# B&R Automation Studio project A2019059_Linka_Power_CP (part 59)

#### Main.st - Cyclic code
```iecst
//******************************************************************************************************
//	Cylic task for recipe management
//
//	Error numbers:
//	50100  Recipe name parameter is empty
//	50101  Recipe name already exists
//	50102  Recipe name was not found
//  50103  One or more recipe names exceeds maximum length
//	50110  Device name parameter is empty
//	50120  Variable name parameter is empty
//  50130  Recipe management is not initialized
//  50200  Maximum number of recipes reached
//  50300  Task name is incorrect
//  50310  Global recipe structure is incorrect
//******************************************************************************************************

//******************************************************************************************************
// Cyclic task
//******************************************************************************************************

PROGRAM _INIT
		// ----------------------------------------------------------------------------------------
	// The following settings can be adjusted
	Recipe_01.PAR.RecipeVariable 	:= 'RecipeData';		// Top variable structure with recipe data
	Recipe_01.PAR.DeviceName 	:= 'HDD_Receptury';		// Device name from the CPU configuration for X20CPU

	// ----------------------------------------------------------------------------------------
	this							:= 'Recipe_01';			// Name of the global variable structure and this task name
	Recipe_01.PAR.RecipeDirectory 	:= 'Receptury';		        	// Directory where the recipes are stored
	IF(REC_RECIPE_TYPE = typeCSV) THEN
		Recipe_01.PAR.MpLink 		:= gRecipeCsv; 		// MpLink from mappRecipe configuration in physical view
	ELSE
		Recipe_01.PAR.MpLink 		:= gRecipeXml; 		// MpLink from mappRecipe configuration in physical view
	END_IF

	// ----------------------------------------------------------------------------------------
	// Dont change anything below this line
	// ----------------------------------------------------------------------------------------

	// ----------------------------------------------------------------------------------------
	// Make sure global variable structure and task name are correct
	taskStatus := ST_ident(ADR(this), taskGroup, ADR(taskID));
	pvStatus := PV_xgetadr(ADR(this), ADR(pvADR), ADR(pvLEN));
	// Connect global and local structure
	IF(pvStatus = 0) THEN
		RECIPE ACCESS pvADR;
		brsmemset(ADR(RECIPE.ERR), 0 , SIZEOF(RECIPE.ERR));
		RECIPE.PAR.Initialized := FALSE;
	END_IF
	RecipeData;

END_PROGRAM

PROGRAM _CYCLIC
	// --------------------------------------------------------------------------------------------------------------------
	// Make sure task name and global structure correct
	IF(pvStatus <> 0) THEN
		RETURN;
	END_IF
	IF(taskStatus <> 0) THEN
		rec_state := CreateError(ADR(RECIPE), ERR_REC_TASK_NAME, "Meno tasku nieje spravne", rec_state);
		RETURN;
	END_IF

	// --------------------------------------------------------------------------------------------------------------------
	// Make sure we dont exceed maximum number of web clients
	IF(RECIPE.PAR.VisuSlotID > REC_MAX_CLIENTS_ID) THEN
		rec_state := CreateError(ADR(RECIPE), ERR_REC_TOO_MANY_CLIENTS, "More than 3 clients try to connect to recipe managment", rec_state);
		RETURN;
	END_IF

	// --------------------------------------------------------------------------------------------------------------------
	// Cyclic function calls
	MpRecipeCsv_0();
	MpRecipeXml_0();

	//**************************************************************************************************
	// Recipe managment state machine
	//**************************************************************************************************
	CASE rec_state OF
		//**********************************************************************************************
		// Wait for command
		//**********************************************************************************************
		REC_WAIT:
			// --------------------------------------------------------------------------------------------------------------------
			// Track filter change and data refresh
			IF ((brwcscmp(ADR(RecipeFilterOld[VisuSlotID]), ADR(RECIPE.VIS[VisuSlotID].RecipeFilter)) <> 0) OR (RecipeNumOld[VisuSlotID] <> RECIPE.DAT.RecipeNum)) THEN
				brsmemset(ADR(RECIPE.VIS[VisuSlotID].RecipeNames), 0, SIZEOF(RECIPE.VIS[VisuSlotID].RecipeNames));
				idy := 0;
				IF(RECIPE.DAT.RecipeNum > 0) THEN
					FOR idx:=0 TO RECIPE.DAT.RecipeNum - 1 DO
						// --------------------------------------------------------------------------------
						// Verify that file name contains filter
						IF (brwcslen(ADR(RECIPE.VIS[VisuSlotID].RecipeFilter)) = 0 OR IsInstrW(ADR(RECIPE.DAT.RecipeNames[idx]), ADR(RECIPE.VIS[VisuSlotID].RecipeFilter))) THEN
							WString2DataProvider(ADR(RECIPE.DAT.RecipeNames[idx]), ADR(tmpWStr1));
							RECIPE.VIS[VisuSlotID].RecipeNames[idy] := tmpWStr1;
							idy := idy + 1;
						END_IF
					END_FOR;
					brwcscpy(ADR(RecipeFilterOld[VisuSlotID]), ADR(RECIPE.VIS[VisuSlotID].RecipeFilter));
				END_IF
				RecipeNumOld[VisuSlotID] := RECIPE.DAT.RecipeNum;
				RECIPE.VIS[VisuSlotID].RecipeNum := idy;
			END_IF
			// Cylce through the client web seesions
			VisuSlotID := VisuSlotID + 1;
			IF(VisuSlotID > REC_MAX_CLIENTS_ID) THEN
				VisuSlotID := 0;
			END_IF

			// --------------------------------------------------------------------------------------------------------------------
			// Disable buttons in visualization when number of recipes is 0
			IF(RECIPE.DAT.RecipeNum = 0) THEN
				RECIPE.PAR.VisuEnableCommand := FALSE;
			ELSE
				RECIPE.PAR.VisuEnableCommand := TRUE;
			END_IF

			// ----------------------------------------------------------------------------------------
			// Reset error reset
			MpRecipeCsv_0.ErrorReset := FALSE;
			MpRecipeXml_0.ErrorReset := FALSE;
			MpRecipeRegPar_0.ErrorReset := FALSE;

			// ----------------------------------------------------------------------------------------
			// Command refresh
			IF (RECIPE.CMD.Init = TRUE) THEN
				// Reset data structure and trigger name refresh for vis
				brsmemset(ADR(RECIPE.DAT), 0, SIZEOF(RECIPE.DAT));
				brsmemset(ADR(RecipeIDs), 0, SIZEOF(RecipeIDs));
				brsmemset(ADR(RecipeNumOld), 16#FF, SIZEOF(RecipeNumOld));
				// Skip variable binding if already initialized
				IF(MpRecipeRegPar_1.PVName <> 0) THEN
					rec_state := REC_READ_DIR;
				ELSE
					// Register recipe name varibale first if unicode is used
					IF(REC_USE_UNICODE) THEN
						rec_state := REC_REG_NAME;
					ELSE
						rec_state := REC_REG_VAR;
					END_IF
				END_IF
				MpRecipeRegPar_1.Enable := FALSE;
				// ----------------------------------------------------------------------------------------
				// Command new recipe
			ELSIF (RECIPE.CMD.New = TRUE AND RECIPE.PAR.RecipeName <> "") THEN
				// Show current state
				animation := WorkingStatus(ADR(RECIPE), ADR("Vytvaram recepturu..."), animation);
				// Verify that we still have space in list
				IF (RECIPE.DAT.RecipeNum > REC_MAX_NUM) THEN
					rec_state := CreateError(ADR(RECIPE), ERR_REC_MAX_NUM, "Maximalny pocet receptur dosiahnuty", rec_state);
					RETURN;
				END_IF
				// Make sure recipe does not already exist
				IF(FindRecName(ADR(RECIPE), RECIPE.PAR.RecipeName) <> REC_DOES_NOT_EXIST) THEN
					tmpWStr1 := "Nazov raceptury ";
					brwcscat(ADR(tmpWStr1), ADR(RECIPE.PAR.RecipeName));
					brwcscat(ADR(tmpWStr1), ADR(" uz existuje"));
					rec_state := CreateError(ADR(RECIPE), ERR_REC_NAME_EXISTS, tmpWStr1, rec_state);
					RETURN;
				END_IF
				// Turn on variable saving, reset selected recipe, copy recipe name to local variable
				MpRecipeRegPar_1.Enable := TRUE;;
				RECIPE.VIS[RECIPE.PAR.VisuSlotID].RecipeSelect := "";
				rec_state := REC_GEN_FILE_NAME;
				// ----------------------------------------------------------------------------------------
				// Command load recipe
			ELSIF (RECIPE.CMD.Load = TRUE AND RECIPE.PAR.RecipeName <> "") THEN
				// Show current state
				animation := WorkingStatus(ADR(RECIPE), ADR("Nahravam recepturu..."), animation);
				// Turn on variable saving, copy recipe name to local variable
				MpRecipeRegPar_1.Enable := TRUE;;
				rec_state := REC_GEN_FILE_NAME;
				// ----------------------------------------------------------------------------------------
				// Command load recipe
			ELSIF (RECIPE.CMD.Save = TRUE AND (RECIPE.PAR.RecipeName <> "" OR RECIPE.PAR.RecipeNameNew <> "")) THEN
				// Show current state
				animation := WorkingStatus(ADR(RECIPE), ADR("Ukladam recepturu..."), animation);
				IF(RECIPE.PAR.RecipeName = "") THEN
					RECIPE.PAR.RecipeName := RECIPE.PAR.RecipeNameNew;
				END_IF
				// Turn on variable saving, copy recipe name to local variable
				MpRecipeRegPar_1.Enable := TRUE;;
				rec_state := REC_GEN_FILE_NAME;
				// ----------------------------------------------------------------------------------------
				// Command delete recipe
			ELSIF (RECIPE.CMD.Delete = TRUE AND RECIPE.PAR.RecipeName <> "") THEN
				// Show current state, copy recipe name to local variable
				animation := WorkingStatus(ADR(RECIPE), ADR("Mazem recepturu..."), animation);
				rec_state := REC_GEN_FILE_NAME;
				// ----------------------------------------------------------------------------------------
				// Rename recipe
			ELSIF (RECIPE.CMD.Rename = TRUE AND RECIPE.PAR.RecipeName <> "" AND RECIPE.PAR.RecipeNameNew <> "") THEN
				// Show current state
				animation := WorkingStatus(ADR(RECIPE), ADR("Premenovavam recepturu..."), animation);
				// Make sure new recipe name does not already exist
				IF(FindRecName(ADR(RECIPE), RECIPE.PAR.RecipeNameNew) <> REC_DOES_NOT_EXIST) THEN
					tmpWStr1 := "Nove meno receptury ";
					brwcscat(ADR(tmpWStr1), ADR(RECIPE.PAR.RecipeNameNew));
					brwcscat(ADR(tmpWStr1), ADR(" uz existuje"));
					rec_state := CreateError(ADR(RECIPE), ERR_REC_NAME_EXISTS, tmpWStr1, rec_state);
					RETURN;
				END_IF
				// Turn on variable saving, reset selected recipe, copy recipe name to local variable
				MpRecipeRegPar_1.Enable := TRUE;
				brsmemset(ADR(RecipeNumOld), 16#FF, SIZEOF(RecipeNumOld));
				RECIPE.VIS[RECIPE.PAR.VisuSlotID].RecipeSelect := "";
				RecipeNameNew := RECIPE.PAR.RecipeNameNew;
				rec_state := REC_GEN_FILE_NAME;
			END_IF
			RecipeName := RECIPE.PAR.RecipeName;

			// ----------------------------------------------------------------------------------------
			// Check parameters
			IF (RECIPE.CMD.Init OR RECIPE.CMD.New OR RECIPE.CMD.Load OR RECIPE.CMD.Save OR RECIPE.CMD.Rename OR RECIPE.CMD.Delete) THEN
				// Make sure recipe mangament was intialized
				IF (NOT RECIPE.CMD.Init AND NOT RECIPE.PAR.Initialized) THEN
					rec_state := CreateError(ADR(RECIPE), ERR_REC_NOT_INITIALIZED, "Receptury nie su zinicializovane", rec_state);
				END_IF
				// Make sure recipe name is valid
				IF((RECIPE.CMD.New OR RECIPE.CMD.Load OR RECIPE.CMD.Save OR RECIPE.CMD.Rename OR RECIPE.CMD.Delete) AND RecipeName = "") THEN
					rec_state := CreateError(ADR(RECIPE), ERR_REC_NAME_EMPTY, "Meno receptury je prazdne", rec_state);
				END_IF
				// Make sure new recipe name is valid
				IF((RECIPE.CMD.Rename) AND RecipeNameNew = "") THEN
					rec_state := CreateError(ADR(RECIPE), ERR_REC_NAME_EMPTY, "Nova receptura je prazdna", rec_state);
				END_IF
				// Make sure device name is valid
				IF(RECIPE.PAR.DeviceName = '') THEN
					rec_state := CreateError(ADR(RECIPE), ERR_REC_DEV_NAME_EMPTY, "Meno zariadenia je prazdne", rec_state);
				END_IF
				// Make sure variable name is valid
				IF(RECIPE.PAR.RecipeVariable = '') THEN
					rec_state := CreateError(ADR(RECIPE), ERR_REC_VAR_NAME_EMPTY, "Meno premennej je prazdne", rec_state);
				END_IF

				RECIPE.PAR.VisuEnableCommand := FALSE;
			END_IF
			//**********************************************************************************************
			// Register recipe name
			//**********************************************************************************************
		REC_REG_NAME:
			// Generate string for local recipe name
			tmpStr1 := this;
			brsstrcat(ADR(tmpStr1), ADR(':RecipeName'));

			MpRecipeRegPar_0.Enable := TRUE;
			MpRecipeRegPar_0.MpLink := ADR(RECIPE.PAR.MpLink);
			MpRecipeRegPar_0.PVName := ADR(tmpStr1);

			// ----------------------------------------------------------------------------------------
			// OK
			IF (NOT MpRecipeRegPar_0.Active AND NOT MpRecipeRegPar_0.Error) THEN
				rec_state := REC_REG_VAR;
				// Error
			ELSIF (MpRecipeRegPar_0.Error) THEN
				rec_state := CreateError(ADR(RECIPE), MpRecipeRegPar_0.StatusID, "Error trying to register recipe name", rec_state);
			END_IF
			//**********************************************************************************************
			// Register variable structure
			//**********************************************************************************************
		REC_REG_VAR:
			MpRecipeRegPar_1.MpLink := ADR(RECIPE.PAR.MpLink);
			MpRecipeRegPar_1.PVName := ADR(RECIPE.PAR.RecipeVariable);

			// ----------------------------------------------------------------------------------------
			// OK
			IF (NOT MpRecipeRegPar_1.Active AND NOT MpRecipeRegPar_1.Error) THEN
				rec_state := REC_CREATE_DIR;
				// Error
			ELSIF (MpRecipeRegPar_1.Error) THEN
				tmpWStr1 := "Error trying to register variable name ";
				brwcsconv(ADR(tmpWStr2), ADR(RECIPE.PAR.RecipeVariable), brwU8toUC);
				brwcscat(ADR(tmpWStr1), ADR(tmpWStr2));
				rec_state := CreateError(ADR(RECIPE), MpRecipeRegPar_1.StatusID, tmpWStr1, rec_state);
			END_IF
			//**********************************************************************************************
			// Create recipe directory
			//**********************************************************************************************
		REC_CREATE_DIR:
			DCreate.enable 	:= 1;
			DCreate.pDevice	:= ADR(RECIPE.PAR.DeviceName);
			DCreate.pName := ADR(RECIPE.PAR.RecipeDirectory);
			DCreate();

			// ----------------------------------------------------------------------------------------
			// OK
			IF (DCreate.status = OK OR DCreate.status = fiERR_DIR_ALREADY_EXIST) THEN
				// Reset command and return to wait state
				rec_state := REC_READ_DIR;
				// Error
			ELSIF (DCreate.status <> ERR_FUB_BUSY) THEN
				rec_state := CreateError(ADR(RECIPE), DCreate.status, "Porucha vytvorenia adresara", rec_state);
			END_IF
			//**********************************************************************************************
			// Read directory information
			//**********************************************************************************************
		REC_READ_DIR:
			// Show current state
			animation := WorkingStatus(ADR(RECIPE), ADR("Nacitavam recepturu..."), animation);
			// ----------------------------------------------------------------------------------------
			// Clear all entrys
			brsmemset(ADR(RECIPE.DAT), 0, SIZEOF(RECIPE.DAT));
			RECIPE.DAT.RecipeNum := 0;
			// ----------------------------------------------------------------------------------------
			// Set values and get device dir
			DInfo.enable 	:= 1;
			DInfo.pDevice	:= ADR(RECIPE.PAR.DeviceName);
			DInfo();

			// ----------------------------------------------------------------------------------------
			// OK
			IF (DInfo.status = OK) THEN
				rec_state := REC_READ_DIR_1;
			ELSIF (DInfo.status = fiERR_DEVICE_MANAGER) THEN
				tmpWStr1 := "Suborovy system ";
				brwcsconv(ADR(tmpWStr2), ADR(RECIPE.PAR.DeviceName), brwU8toUC);
				brwcscat(ADR(tmpWStr1), ADR(tmpWStr2));
				brwcscat(ADR(tmpWStr1), ADR(" je nedostupny"));
				rec_state := CreateError(ADR(RECIPE), DInfo.status, tmpWStr1, rec_state);
			ELSIF (DInfo.status = fiERR_DIR_NOT_EXIST) THEN
				tmpWStr1 := "Subor ";
				brwcsconv(ADR(tmpWStr2), ADR(RECIPE.PAR.RecipeDirectory), brwU8toUC);
				brwcscat(ADR(tmpWStr1), ADR(tmpWStr2));
				brwcscat(ADR(tmpWStr1), ADR(" je nedostupny"));
				rec_state := CreateError(ADR(RECIPE), DInfo.status, tmpWStr1, rec_state);
				// Error
			ELSIF (DInfo.status <> ERR_FUB_BUSY) THEN
				rec_state := CreateError(ADR(RECIPE), DInfo.status, "Error dir info", rec_state);
			END_IF
			//**********************************************************************************************
			// Open directory
			//**********************************************************************************************
		REC_READ_DIR_1:
			DOpen.enable 	:= 1;
			DOpen.pDevice	:= ADR(RECIPE.PAR.DeviceName);
			DOpen.pName 	:= ADR(RECIPE.PAR.RecipeDirectory);
			DOpen();

			// ----------------------------------------------------------------------------------------
			// OK
			IF (DOpen.status = OK) THEN
				rec_state := REC_READ_DIR_2;
			ELSIF (DInfo.status = fiERR_DIR_NOT_EXIST) THEN
				tmpWStr1 := "Adresar ";
				brwcsconv(ADR(tmpWStr2), ADR(RECIPE.PAR.RecipeDirectory), brwU8toUC);
				brwcscat(ADR(tmpWStr1), ADR(tmpWStr2));
				brwcscat(ADR(tmpWStr1), ADR(" je nedostupny"));
				rec_state := CreateError(ADR(RECIPE), DInfo.status, tmpWStr1, rec_state);
				// Error
			ELSIF (DOpen.status <> ERR_FUB_BUSY) THEN
				rec_state := CreateError(ADR(RECIPE), DOpen.status, "Porucha otvorenie adresara", rec_state);
			END_IF;
			//**********************************************************************************************
			// Read file directory information
			//**********************************************************************************************
		REC_READ_DIR_2:
			DRead.enable 	:= 1;
			DRead.ident		:= DOpen.ident;
			DRead.pData 	:= ADR(lDirReadData);
			DRead.data_len 	:= SIZEOF(lDirReadData);
			DRead();

			// ----------------------------------------------------------------------------------------
			// OK
			IF (DRead.status = OK AND lDirReadData.Mode = fiFILE) THEN
				animation := WorkingStatus(ADR(RECIPE), ADR("Inicializacia receptur..."), animation);
				// Make sure file name does not exceed maximum string size
				IF (brsstrlen(ADR(lDirReadData.Filename)) < REC_NAME_LENGTH) THEN
					// Copy dir info to string
					brsmemset(ADR(RECIPE.PAR.RecipeID), 0, SIZEOF(RECIPE.PAR.RecipeID));
					brsstrcpy(ADR(RECIPE.PAR.RecipeID), ADR(lDirReadData.Filename));
					// Make sure file extension is CSV or XML
					IF(brsstrlen(ADR(RECIPE.PAR.RecipeID)) > 4 AND ((REC_RECIPE_TYPE = typeCSV AND brsmemcmp(ADR(RECIPE.PAR.RecipeID) + (brsstrlen(ADR(RECIPE.PAR.RecipeID)) - 4), ADR('.csv'), 4) = 0) OR (REC_RECIPE_TYPE = typeXML AND brsmemcmp(ADR(RECIPE.PAR.RecipeID) + (brsstrlen(ADR(RECIPE.PAR.RecipeID)) - 4), ADR('.xml'), 4) = 0))) THEN
						brsmemset(ADR(RECIPE.PAR.RecipeID) + (brsstrlen(ADR(RECIPE.PAR.RecipeID)) - 4), 0, 4);
						// ------------------------------------------------------------------------------------
						// Verify that we still have space in list
						IF (RECIPE.DAT.RecipeNum <= REC_MAX_NUM) THEN
							// --------------------------------------------------------------------
							// Read recipe name from recipe data in next step when using unicode
							IF(REC_USE_UNICODE) THEN
								RecipeIDs[brsatoi(ADR(RECIPE.PAR.RecipeID))] := TRUE;
								rec_state := REC_GEN_FILE_NAME;
								// Generate recipe name from file name
							ELSE
								brwcsconv(ADR(RecipeName), ADR(RECIPE.PAR.RecipeID), brwU8toUC);
								// Generate ASCII data, insert recipe into list
								InsertRecName(ADR(RECIPE), RecipeName, RECIPE.PAR.RecipeID);
							END_IF
							// Error
						ELSE
							rec_state := CreateError(ADR(RECIPE), ERR_REC_MAX_NUM, "Maximalny pocet receptur dosiahnuty", rec_state);
						END_IF
					END_IF
				ELSE
					has_oversized_items := TRUE;
				END_IF
				// Last entry reached
			ELSIF (DRead.status = fiERR_NO_MORE_ENTRIES) THEN
				rec_state := REC_READ_DIR_3;
				// Error
			ELSIF (DRead.status <> ERR_FUB_BUSY AND DRead.status <> OK) THEN
				rec_state := CreateError(ADR(RECIPE), DRead.status, "Porucha citania zoznamu receptur", rec_state);
			END_IF
			//**********************************************************************************************
			// Close directory information
			//**********************************************************************************************
		REC_READ_DIR_3:
			DClose.enable 	:= 1;
			DClose.ident	:= DOpen.ident;
			DClose();

			// ----------------------------------------------------------------------------------------
			// OK
			IF (DClose.status = OK) THEN
				// Reset command and return to wait state
				RECIPE.DAT.Status := "Inicializacia receptur ukoncena";
				RECIPE.CMD.Init	:= 0;
				RECIPE.PAR.RecipeID := '';
				RECIPE.PAR.Initialized := TRUE;
				DClose.ident	:= 0;
				IF(has_oversized_items) THEN
					rec_state := CreateError(ADR(RECIPE), ERR_REC_NAME_LENGTH, "Meno receptury presiahlo maximalny pocet znakov", rec_state);
				ELSE
					rec_state := REC_WAIT;
				END_IF
				// Error
			ELSIF (DClose.status <> ERR_FUB_BUSY) THEN
				rec_state := CreateError(ADR(RECIPE), DClose.status, "Porucha zatvorenia adresara", rec_state);
			END_IF
			//**********************************************************************************************
			// Generate recipe name	full path and file name
			//**********************************************************************************************
		REC_GEN_FILE_NAME:
			// Find recipe entry
			RecipeIndex := FindRecName(ADR(RECIPE), RecipeName);

			// Generate file name when using unicode strings
			IF(REC_USE_UNICODE) THEN
				// Ignore during init process
				IF(NOT RECIPE.CMD.Init) THEN
					// Find empty slot for new recipe
					IF(RECIPE.CMD.New) THEN
						RecipeIndex := 0;
						WHILE (RecipeIDs[RecipeIndex] = TRUE AND RecipeIndex <= REC_MAX_NUM) DO
							RecipeIndex := RecipeIndex + 1;
						END_WHILE;
						// Make sure we found empty slot
						IF(RecipeIndex <= REC_MAX_NUM AND RecipeIDs[RecipeIndex] = FALSE) THEN
							brsitoa(RecipeIndex, ADR(RECIPE.PAR.RecipeID));
						ELSE
							rec_state := CreateError(ADR(RECIPE), ERR_REC_MAX_NUM, "Prazdny slot nenajdeny", rec_state);
							RETURN;
						END_IF
						// Find recipe name in list	for all other command
					ELSE
						// Recipe name was found
						IF(RecipeIndex <> REC_DOES_NOT_EXIST) THEN
							RECIPE.PAR.RecipeID := RECIPE.DAT.RecipeIDs[RecipeIndex];
							// Recipe name was lost
						ELSE
							tmpWStr1 := "Meno receptury nebolo najdene ";
							brwcscat(ADR(tmpWStr1), ADR(RecipeName));
							rec_state := CreateError(ADR(RECIPE), ERR_REC_NAME_LOST, tmpWStr1, rec_state);
							RETURN;
						END_IF
					END_IF
				END_IF
				// Use recipe name as file name when using standard strings
			ELSE
				brwcsconv(ADR(RECIPE.PAR.RecipeID), ADR(RecipeName), brwUCtoU8);
			END_IF

			// Generate recipe path and extension
			RecipeFullFileName := RECIPE.PAR.RecipeDirectory;
			brsstrcat(ADR(RecipeFullFileName), ADR('/'));
			brsstrcat(ADR(RecipeFullFileName), ADR(RECIPE.PAR.RecipeID));

			// Add file extension
			IF(REC_RECIPE_TYPE = typeCSV) THEN
				brsstrcat(ADR(RecipeFullFileName), ADR('.csv'));
			ELSE
				brsstrcat(ADR(RecipeFullFileName), ADR('.xml'));
			END_IF

			// Save recipe under new name
			IF(RECIPE.CMD.Rename) THEN
				RecipeName := RecipeNameNew;
			END_IF

			// Proceed with next step
			IF(RECIPE.CMD.Delete) THEN
				rec_state := REC_DELETE;
			ELSIF(RECIPE.CMD.Rename AND NOT REC_USE_UNICODE) THEN
				rec_state := REC_RENAME;
			ELSE
				rec_state := REC_LOAD_SAVE;
			END_IF
			//**********************************************************************************************
			// Load or save recipe data
			//**********************************************************************************************
		REC_LOAD_SAVE:

			IF(REC_RECIPE_TYPE = typeCSV) THEN
				MpRecipeCsv_0.Enable := TRUE;
				MpRecipeCsv_0.MpLink := ADR(RECIPE.PAR.MpLink);
				MpRecipeCsv_0.DeviceName := ADR(RECIPE.PAR.DeviceName);
				MpRecipeCsv_0.FileName := ADR(RecipeFullFileName);
				MpRecipeCsv_0.Save := RECIPE.CMD.Save OR RECIPE.CMD.New OR RECIPE.CMD.Rename;
				MpRecipeCsv_0.Load := RECIPE.CMD.Load OR RECIPE.CMD.Init;

				MpRecipeDone := MpRecipeCsv_0.CommandDone;
				MpRecipeError := MpRecipeCsv_0.Error;
				MpRecipeStatusID := MpRecipeCsv_0.StatusID;
			ELSE
				MpRecipeXml_0.Enable := TRUE;
				MpRecipeXml_0.MpLink := ADR(RECIPE.PAR.MpLink);
				MpRecipeXml_0.DeviceName := ADR(RECIPE.PAR.DeviceName);
				MpRecipeXml_0.FileName := ADR(RecipeFullFileName);
				MpRecipeXml_0.Save := RECIPE.CMD.Save OR RECIPE.CMD.New OR RECIPE.CMD.Rename;
				MpRecipeXml_0.Load := RECIPE.CMD.Load OR RECIPE.CMD.Init;

				MpRecipeDone := MpRecipeXml_0.CommandDone;
				MpRecipeError := MpRecipeXml_0.Error;
				MpRecipeStatusID := MpRecipeXml_0.StatusID;
			END_IF

			// ----------------------------------------------------------------------------------------
			// OK
			IF (MpRecipeDone AND NOT MpRecipeError AND MpRecipeStatusID = 0) THEN
				// Reset command and return to wait state
				MpRecipeCsv_0.Load := FALSE;
				MpRecipeCsv_0.Save := FALSE;
				MpRecipeXml_0.Load := FALSE;
				MpRecipeXml_0.Save := FALSE;

				// Continue renaming recipe
				IF(RECIPE.CMD.Rename) THEN
					IF(REC_USE_UNICODE) THEN
						// Remove name from recipe list	and add it again
						RemoveRecName(ADR(RECIPE), RecipeIndex);
						InsertRecName(ADR(RECIPE), RecipeName, RECIPE.PAR.RecipeID);

						RECIPE.VIS[RECIPE.PAR.VisuSlotID].RecipeSelect := RecipeName;
						tmpWStr1 := "Receptura bola premenovana";
						RECIPE.CMD.Rename := 0;
					ELSE
						rec_state := REC_DELETE;
						RETURN;
					END_IF
				END_IF
				// Continue reading recipe names
				IF(RECIPE.CMD.Init) THEN
					InsertRecName(ADR(RECIPE), RecipeName, RECIPE.PAR.RecipeID);
					rec_state := REC_READ_DIR_2;
					RETURN;
				END_IF
				// Finish new recipe
				IF(RECIPE.CMD.New) THEN
					IF(REC_USE_UNICODE) THEN
						RecipeIDs[brsatoi(ADR(RECIPE.PAR.RecipeID))] := TRUE;
					END_IF
					InsertRecName(ADR(RECIPE), RecipeName, RECIPE.PAR.RecipeID);
					RECIPE.VIS[RECIPE.PAR.VisuSlotID].RecipeSelect := RecipeName;
					tmpWStr1 := "Receptura bola vytvorena";
					RECIPE.CMD.New	:= FALSE;
				END_IF
				// Finish load recipe
				IF(RECIPE.CMD.Load) THEN
					tmpWStr1 := "Receptura bola nacitana";
					RECIPE.CMD.Load	:= FALSE;
				END_IF
				// Finish save recipe
				IF(RECIPE.CMD.Save) THEN
					tmpWStr1 := "Receptura bola ulozena";
					RECIPE.CMD.Save	:= FALSE;
				END_IF
				// Complete status string
				CreateMessage(ADR(RECIPE.DAT.Status), ADR(tmpWStr1), ADR(RecipeName), RECIPE.PAR.VisuSlotID);
				rec_state := REC_WAIT;
				// Error
			ELSIF (MpRecipeStatusID = mpRECIPE_WRN_LOAD_WITH_WARN) THEN
				rec_state := CreateError(ADR(RECIPE), MpRecipeStatusID, "Warning recipe read/write/new, check PLC logbook for details", rec_state);
			ELSIF (MpRecipeError OR MpRecipeStatusID <> 0) THEN
				tmpWStr1 := "Error recipe read/write/new ";
				brwcscat(ADR(tmpWStr1), ADR(RecipeName));
				rec_state := CreateError(ADR(RECIPE), MpRecipeStatusID, tmpWStr1, rec_state);
			END_IF
			//**********************************************************************************************
			// Delete selected recipe
			//**********************************************************************************************
		REC_DELETE:
			// ----------------------------------------------------------------------------------------
			// Initialize file delete structure
			FDelete.enable		:= 1;
			FDelete.pDevice 	:= ADR(RECIPE.PAR.DeviceName);
			FDelete.pName		:= ADR(RecipeFullFileName);
			FDelete();

			// ----------------------------------------------------------------------------------------
			// OK
			IF (FDelete.status = OK) THEN
				// Remove name from recipe list
				RemoveRecName(ADR(RECIPE), RecipeIndex);
				// Mark recipe ID as free
				IF(REC_USE_UNICODE) THEN
					RecipeIDs[brsatoi(ADR(RECIPE.PAR.RecipeID))] := FALSE;
				END_IF

				CreateMessage(ADR(RECIPE.DAT.Status), ADR("Receptura bola vymazana"), ADR(RecipeName), RECIPE.PAR.VisuSlotID);
				RECIPE.CMD.Delete := 0;
				rec_state := REC_WAIT;
				// Error
			ELSIF (FDelete.status <> ERR_FUB_BUSY) THEN
				tmpWStr1 := "Porucha vymazania receptury ";
				brwcscat(ADR(tmpWStr1), ADR(RecipeName));
				rec_state := CreateError(ADR(RECIPE), FDelete.status, tmpWStr1, rec_state);
			END_IF
			//**********************************************************************************************
			// Rename selected recipe
			//**********************************************************************************************
		REC_RENAME:
			// Generate recipe path and extension
			tmpStr1 := RECIPE.PAR.RecipeDirectory;
			brsstrcat(ADR(tmpStr1), ADR('/'));
			brwcsconv(ADR(tmpStr2), ADR(RecipeNameNew), brwUCtoU8);
			brsstrcat(ADR(tmpStr1), ADR(tmpStr2));

			// Add file extension
			IF(REC_RECIPE_TYPE = typeCSV) THEN
				brsstrcat(ADR(tmpStr1), ADR('.csv'));
			ELSE
				brsstrcat(ADR(tmpStr1), ADR('.xml'));
			END_IF

			// ----------------------------------------------------------------------------------------
			// Initialize file delete structure
			FRename.enable		:= 1;
			FRename.pDevice 	:= ADR(RECIPE.PAR.DeviceName);
			FRename.pName		:= ADR(RecipeFullFileName);
			FRename.pNewName	:= ADR(tmpStr1);
			FRename();

			// ----------------------------------------------------------------------------------------
			// OK
			IF (FRename.status = OK) THEN
				// Remove name from recipe list	and add it again
				brsmemmove(ADR(RECIPE.DAT.RecipeNames[RecipeIndex]),ADR(RECIPE.DAT.RecipeNames[RecipeIndex+1]), (RECIPE.DAT.RecipeNum) * SIZEOF(RECIPE.DAT.RecipeNames[0]));
				brsmemmove(ADR(RECIPE.DAT.RecipeIDs[RecipeIndex]),ADR(RECIPE.DAT.RecipeIDs[RecipeIndex+1]), (RECIPE.DAT.RecipeNum) * SIZEOF(RECIPE.DAT.RecipeIDs[0]));
				RECIPE.DAT.RecipeNum := RECIPE.DAT.RecipeNum - 1;
				InsertRecName(ADR(RECIPE), RecipeNameNew, RECIPE.PAR.RecipeID);

				RECIPE.VIS[RECIPE.PAR.VisuSlotID].RecipeSelect := RecipeNameNew;
				CreateMessage(ADR(RECIPE.DAT.Status), ADR("Receptura bola premenovana"), ADR(RecipeName), RECIPE.PAR.VisuSlotID);
				RECIPE.CMD.Rename := 0;
				rec_state := REC_WAIT;
				// Error
			ELSIF (FRename.status <> ERR_FUB_BUSY) THEN
				tmpWStr1 := "Porucha premenovania receptury ";
				brwcscat(ADR(tmpWStr1), ADR(RecipeName));
				rec_state := CreateError(ADR(RECIPE), FRename.status, tmpWStr1, rec_state);
			END_IF
			// --------------------------------------------------------------------------------------------------------------------
			// Error
			// --------------------------------------------------------------------------------------------------------------------
		REC_ERROR:
			RECIPE.DAT.Status := "Error state triggered on web client ID ";
			tmpWStr1 := DINT_TO_WSTRING(RECIPE.PAR.VisuSlotID);
			brwcscat(ADR(RECIPE.DAT.Status), ADR(tmpWStr1));
			// --------------------------------------------------------------------------------------------------------------------
			// Make sure we dont exceed maximum number of web clients
			IF(RECIPE.PAR.VisuSlotID <= REC_MAX_CLIENTS_ID) THEN
				RECIPE.VIS[RECIPE.PAR.VisuSlotID].ShowMessageBoxError := TRUE;
			END_IF
			// --------------------------------------------------------------------------------------------------------------------
			// Return to idle state
			IF RECIPE.CMD.ErrorReset THEN
				// Reset function blocks
				MpRecipeCsv_0.ErrorReset := TRUE;
				MpRecipeCsv_0.Save := FALSE;
				MpRecipeCsv_0.Load := FALSE;

				MpRecipeXml_0.ErrorReset := TRUE;
				MpRecipeXml_0.Save := FALSE;
				MpRecipeXml_0.Load := FALSE;

				MpRecipeRegPar_0.ErrorReset := TRUE;

				// Reset error structure
				brsmemset(ADR(RECIPE.ERR), 0, SIZEOF(RECIPE.ERR));
				RECIPE.DAT.Status := "";
				RECIPE.CMD.ErrorReset := FALSE;
				RECIPE.VIS[RECIPE.PAR.VisuSlotID].ShowMessageBoxError := FALSE;
				rec_state := REC_WAIT;
			END_IF;
			brsmemset(ADR(RECIPE.CMD), 0, SIZEOF(RECIPE.CMD));
			RETURN;
	END_CASE
	// --------------------------------------------------------------------------------------------------------------------
	// Cyclic function calls
	MpRecipeRegPar_0();
	MpRecipeRegPar_1();
	MpRecipeCsv_0();
	MpRecipeXml_0();

END_PROGRAM

PROGRAM _EXIT
	(* Insert code here *)

END_PROGRAM
```

#### RecipeVariables.var - Local variables
```iecst
(*------------------------------------------------------------------------------------------------------------------------------------------------------------------------------------------------------------------------*)
(*Local constants*)
VAR CONSTANT
	OK : USINT := 0; (*Constant for status OK *)
	REC_DOES_NOT_EXIST : UINT := 65535; (*Constant for record does not exist*)
END_VAR
(*------------------------------------------------------------------------------------------------------------------------------------------------------------------------------------------------------------------------*)
(*Local Variables*)
VAR
	RECIPE : REFERENCE TO recMAIN; (*Local recipe structure*)
	RecipeIDs : ARRAY[0..REC_MAX_NUM] OF BOOL; (*Used with unicode option, keeps tracks of the IDs used*)
	RecipeIndex : UINT; (*Current recipe index*)
	RecipeName : WSTRING[REC_NAME_LENGTH]; (*Local recipe name*)
	RecipeNameNew : WSTRING[REC_NAME_LENGTH]; (*Local recipe new name*)
	RecipeFullFileName : STRING[200]; (*Full recipe name*)
	RecipeFilterOld : ARRAY[0..REC_MAX_CLIENTS_ID] OF WSTRING[REC_NAME_LENGTH]; (*Track filter change *)
	RecipeNumOld : ARRAY[0..REC_MAX_CLIENTS_ID] OF UINT;
	rec_state : recSTATE := REC_WAIT; (*Main step index *)
	animation : USINT := 0; (*Animation for working status	*)
	VisuSlotID : USINT; (*Slot of the visualization that is current used*)
	idx : UINT;
	idy : UINT;
	has_oversized_items : BOOL; (*Indicates that at least one recipe name exceeds the maximum length*)
	tmpStr1 : STRING[200]; (*Temporary string variable *)
	tmpStr2 : STRING[200]; (*Temporary string variable *)
	tmpWStr1 : WSTRING[REC_VIS_LENGTH]; (*Temporary unicode string variable *)
	tmpWStr2 : WSTRING[REC_VIS_LENGTH]; (*Temporary unicode string variable *)
	lDirReadData : fiDIR_READ_EX_DATA; (*File information structure*)
	this : STRING[100]; (*Name of the task and global recipe structure*)
	taskID : UDINT; (*Task ID*)
	taskGroup : USINT; (*Task Group*)
	taskStatus : UINT; (*Status of task information*)
	pvADR : UDINT; (*Adress of global variable structure*)
	pvLEN : UDINT; (*Lenght of global variable structure*)
	pvStatus : UINT; (*Status of global variable information*)
	MpRecipeDone : BOOL; (*Generic status done*)
	MpRecipeError : BOOL; (*Genereic status error*)
	MpRecipeStatusID : DINT; (*Generic error details*)
END_VAR
(*------------------------------------------------------------------------------------------------------------------------------------------------------------------------------------------------------------------------*)
(*Local function calls*)
VAR
	DInfo : DirInfo;
	DOpen : DirOpen;
	DRead : DirReadEx;
	DClose : DirClose;
	DCreate : DirCreate;
	FDelete : FileDelete;
	FRename : FileRename;
	MpRecipeCsv_0 : MpRecipeCsv;
	MpRecipeXml_0 : MpRecipeXml;
	MpRecipeRegPar_0 : MpRecipeRegPar;
	MpRecipeRegPar_1 : MpRecipeRegPar;
END_VAR
(*------------------------------------------------------------------------------------------------------------------------------------------------------------------------------------------------------------------------*)
(*Error numbers*)
VAR CONSTANT
	ERR_REC_TOO_MANY_CLIENTS : DINT := 50010; (*More than 3 clients try to connect to recipe management*)
	ERR_REC_NAME_EMPTY : DINT := 50100; (*Recipe name is empty*)
	ERR_REC_NAME_EXISTS : DINT := 50101; (*Recipe name already exists*)
	ERR_REC_NAME_LOST : DINT := 50102; (*Recipe name was not found*)
	ERR_REC_NAME_LENGTH : DINT := 50103; (*One or more recipe names exceeds maximum length*)
	ERR_REC_DEV_NAME_EMPTY : DINT := 50110; (*Device name is empty*)
	ERR_REC_VAR_NAME_EMPTY : DINT := 50120; (*Variable name is empty*)
	ERR_REC_NOT_INITIALIZED : DINT := 50130; (*Recipemanagement is not initialized*)
	ERR_REC_MAX_NUM : DINT := 50200; (*Maximum number of recipes reached*)
	ERR_REC_TASK_NAME : DINT := 50300; (*Task name is incorrect*)
	ERR_REC_GLOBAL_VAR : DINT := 50231; (*Maximum number of recipes reached*)
END_VAR
```

#### LocalFunctions.fun - Local function definition
```iecst
FUNCTION CreateError : recSTATE
	VAR_INPUT
		RECIPE : REFERENCE TO recMAIN;
		No : DINT;
		Text : WSTRING[200];
		State : recSTATE;
	END_VAR
END_FUNCTION

FUNCTION CreateMessage : BOOL
	VAR_INPUT
		TargetString : UDINT;
		Text : UDINT;
		RecipeName : UDINT;
		VisuSlotID : USINT;
	END_VAR
	VAR
		VisuSlotIDStr : WSTRING[5];
		tmpWStr1 : WSTRING[200];
	END_VAR
END_FUNCTION

FUNCTION FindRecName : UINT
	VAR_INPUT
		RECIPE : REFERENCE TO recMAIN;
		RecipeName : WSTRING[REC_NAME_LENGTH];
	END_VAR
	VAR
		idx : UINT;
	END_VAR
END_FUNCTION

FUNCTION InsertRecName : UINT
	VAR_INPUT
		RECIPE : REFERENCE TO recMAIN;
		new_name : WSTRING[REC_NAME_LENGTH];
		new_id : STRING[REC_NAME_LENGTH];
	END_VAR
	VAR
		idx : INT;
		idy : INT;
		lSort : DINT;
	END_VAR
END_FUNCTION

FUNCTION RemoveRecName : BOOL
	VAR_INPUT
		RECIPE : REFERENCE TO recMAIN;
		RecipeIndex : UINT;
	END_VAR
END_FUNCTION

FUNCTION IsInstrW : BOOL
	VAR_INPUT
		string1 : UDINT;
		string2 : UDINT;
	END_VAR
	VAR
		idx : UDINT;
	END_VAR
END_FUNCTION

FUNCTION WorkingStatus : USINT
	VAR_INPUT
		RECIPE : REFERENCE TO recMAIN;
		str : UDINT;
		animation : USINT;
	END_VAR
END_FUNCTION

FUNCTION WString2DataProvider : BOOL
	VAR_INPUT
		SourceString : UDINT;
		TargetString : UDINT;
	END_VAR
END_FUNCTION
```

#### LocalFunctions.st - Local function code
```iecst
//******************************************************************************************************
// Find recipe name
//******************************************************************************************************
FUNCTION FindRecName
	// Check if recipe name exists
	IF(RECIPE.DAT.RecipeNum > 0) THEN
		FOR idx:=0 TO RECIPE.DAT.RecipeNum - 1 DO
			IF(RECIPE.DAT.RecipeNames[idx] = RecipeName) THEN
				FindRecName := idx;
				RETURN;
			END_IF
		END_FOR;
	END_IF
	FindRecName := REC_DOES_NOT_EXIST;
END_FUNCTION

//******************************************************************************************************
// Create mappView data provider string
//******************************************************************************************************
FUNCTION WString2DataProvider
	brwcscpy(TargetString, ADR("{$"value$":$""));
	brwcscat(TargetString, SourceString);
	brwcscat(TargetString, ADR("$",$"text$":$""));
	brwcscat(TargetString, SourceString);
	brwcscat(TargetString, ADR("$"}"));

	WString2DataProvider := TRUE;
END_FUNCTION

//******************************************************************************************************
// Create error
//******************************************************************************************************
FUNCTION CreateError
	RECIPE.ERR.No := No;
	RECIPE.ERR.State := State;
	RECIPE.ERR.Text := Text;
	CreateError := REC_ERROR;
END_FUNCTION

//******************************************************************************************************
// Create status meesage
//******************************************************************************************************
FUNCTION CreateMessage
	brwcscpy(ADR(tmpWStr1), Text);
	brwcscat(ADR(tmpWStr1), ADR(" "));
	brwcscat(ADR(tmpWStr1), RecipeName);
	brwcscat(ADR(tmpWStr1), ADR(" on web client ID "));
	VisuSlotIDStr := DINT_TO_WSTRING(VisuSlotID);
	brwcscat(ADR(tmpWStr1), ADR(VisuSlotIDStr));
	brwcscpy(TargetString, ADR(tmpWStr1));

	CreateMessage := TRUE;
END_FUNCTION

//******************************************************************************************************
// Working status
//******************************************************************************************************
FUNCTION WorkingStatus
	animation := animation+1;

	IF (animation = 80) THEN
		animation := 0;
	END_IF

	brsmemset(ADR(RECIPE.DAT.Status), 0, SIZEOF(RECIPE.DAT.Status));
	brwcscpy(ADR(RECIPE.DAT.Status), str);
	CASE(animation) OF
		0..19	: brwcscat(ADR(RECIPE.DAT.Status), ADR("/"));
		20..39	: brwcscat(ADR(RECIPE.DAT.Status), ADR("-"));
		40..59	: brwcscat(ADR(RECIPE.DAT.Status), ADR("\"));
		60..79	: brwcscat(ADR(RECIPE.DAT.Status), ADR("|"));
	END_CASE;
	WorkingStatus := animation;
END_FUNCTION

//******************************************************************************************************
// Fill new folder or directory name
//******************************************************************************************************
FUNCTION RemoveRecName
	// Remove name from recipe list
	IF(RecipeIndex < REC_MAX_NUM) THEN
		brsmemmove(ADR(RECIPE.DAT.RecipeNames[RecipeIndex]),ADR(RECIPE.DAT.RecipeNames[RecipeIndex+1]), (REC_MAX_NUM - RecipeIndex) * SIZEOF(RECIPE.DAT.RecipeNames[0]));
		brsmemmove(ADR(RECIPE.DAT.RecipeIDs[RecipeIndex]),ADR(RECIPE.DAT.RecipeIDs[RecipeIndex+1]), (REC_MAX_NUM - RecipeIndex) * SIZEOF(RECIPE.DAT.RecipeIDs[0]));
	END_IF
	brsmemset(ADR(RECIPE.DAT.RecipeNames[REC_MAX_NUM]), 0, SIZEOF(ADR(RECIPE.DAT.RecipeNames[0])));
	brsmemset(ADR(RECIPE.DAT.RecipeIDs[REC_MAX_NUM]), 0, SIZEOF(ADR(RECIPE.DAT.RecipeIDs[0])));
	RECIPE.DAT.RecipeNum := RECIPE.DAT.RecipeNum - 1;
	RemoveRecName := TRUE;
END_FUNCTION

//******************************************************************************************************
// Fill new folder or directory name
//******************************************************************************************************
FUNCTION InsertRecName
	// Set up start values for iteration
	IF (RECIPE.DAT.RecipeNum <> 0) THEN
		idy := RECIPE.DAT.RecipeNum - 1;
	END_IF
	idx := idy;

	// Start iteration	search
	WHILE (idy > 1) DO
		// Check current entry
		lSort := brwcscmp(ADR(new_name), ADR(RECIPE.DAT.RecipeNames[idy]));
		// Solve new search range
		IF (idy MOD 2 = 0) THEN
			idy := idy / 2;
		ELSE
			idy := idy / 2 + 1;
		END_IF
		// New range is lower or higher than current
		IF (lSort > 0) THEN
			idx := idx + idy;
			IF (idx > UINT_TO_INT(RECIPE.DAT.RecipeNum)) THEN
				idx := RECIPE.DAT.RecipeNum;
			END_IF
		ELSE
			idx := idx - idy;
			IF (idx < 1) THEN
				idx := 1;
			END_IF
		END_IF
	END_WHILE;

	// New entry is this, next or previous
	lSort := brwcscmp(ADR(new_name), ADR(RECIPE.DAT.RecipeNames[idx]));
	IF (lSort > 0 AND idx <> UINT_TO_INT(RECIPE.DAT.RecipeNum)) THEN
		idx := idx +1;
	ELSIF (idx > 0) THEN
		lSort := brwcscmp(ADR(new_name), ADR(RECIPE.DAT.RecipeNames[idx-1]));
		IF (lSort < 0) THEN
			idx := idx - 1;
		END_IF
	END_IF

	// Move all data entrys backwards and fill in new entry
	IF(idx < REC_MAX_NUM) THEN
		brsmemmove(ADR(RECIPE.DAT.RecipeNames[idx+1]),ADR(RECIPE.DAT.RecipeNames[idx]), (RECIPE.DAT.RecipeNum - idx) * SIZEOF(RECIPE.DAT.RecipeNames[1]));
		brsmemmove(ADR(RECIPE.DAT.RecipeIDs[idx+1]),ADR(RECIPE.DAT.RecipeIDs[idx]), (RECIPE.DAT.RecipeNum - idx) * SIZEOF(RECIPE.DAT.RecipeIDs[1]));
	END_IF
	brwcscpy(ADR(RECIPE.DAT.RecipeNames[idx]), ADR(new_name));
	brsstrcpy(ADR(RECIPE.DAT.RecipeIDs[idx]), ADR(new_id));

	RECIPE.DAT.RecipeNum := RECIPE.DAT.RecipeNum + 1;
	InsertRecName := idx;
END_FUNCTION

//******************************************************************************************************
// Is second string in first string
//******************************************************************************************************
FUNCTION IsInstrW
	IF (brwcslen(string1) >= brwcslen(string2)) THEN
		FOR idx:=0 TO brwcslen(string1) - brwcslen(string2) DO
			IF (brwcsncmp(string1 + idx, string2, brwcslen(string2)) = 0) THEN
				IsInstrW := TRUE;
				EXIT;
			END_IF
		END_FOR;
	END_IF
END_FUNCTION
```

### UsersGlobal.typ - Global data types
```iecst
TYPE
	UsersVizu_typ : 	STRUCT
		TypPrihlasenia : USINT;
		ZoznamUzivatelov : ARRAY[0..100]OF STRING[100];
		Edit_MenoUzivatela : STRING[80]; (*Meno zadavané pri uložení uživatela*)
		Edit_HesloUzivatela : STRING[80]; (*Heslo zadané pri uložení uživatela*)
		Edit_CisloKarty : STRING[80]; (*Cislo karty nacitane pri uložení uživatela*)
		Edit_UrovenUzivatela : STRING[80];
		CisloPrihlasenejKarty_Panel1 : STRING[80]; (*Cislo karty nacitane pri uložení uživatela*)
		CisloPrihlasenejKarty_Panel2 : STRING[80]; (*Cislo karty nacitane pri uložení uživatela*)
		CisloPrihlasenejKarty_Panel3 : STRING[80]; (*Cislo karty nacitane pri uložení uživatela*)
		ZadaneMenoUzivatela : STRING[80]; (*Meno zadané cez prihlasovacie okno*)
		ZadaneHesloUzivatela : STRING[80]; (*Heslo zadané cez prihlasovacie okno*)
		ZadaneCisloKarty_Panel1 : STRING[80]; (*Cislo karty načítané pri prihlásení*)
		ZadaneCisloKarty_Panel2 : STRING[80]; (*Cislo karty načítané pri prihlásení*)
		ZadaneCisloKarty_Panel3 : STRING[80]; (*Cislo karty načítané pri prihlásení*)
		MenoPrihlasenehoUzivatela_Panel1 : STRING[80]; (*Zobrazuje sa vo vizualizácii*)
		MenoPrihlasenehoUzivatela_Panel2 : STRING[80]; (*Zobrazuje sa vo vizualizácii*)
		MenoPrihlasenehoUzivatela_Panel3 : STRING[80]; (*Zobrazuje sa vo vizualizácii*)
		UlozUzivatela : BOOL;
		PrihlasUzivatela : BOOL;
		VymazUzivatela : BOOL;
		OdhlasUzivatela_Panel1 : BOOL;
		OdhlasUzivatela_Panel2 : BOOL;
		OdhlasUzivatela_Panel3 : BOOL;
		NacitajUzivatela : BOOL;
		LB_Index : UINT;
		LB_IndexSTRING : STRING[80];
		KartaPrilozena_Panel1 : BOOL;
		KartaPrilozena_Panel2 : BOOL;
		KartaPrilozena_Panel3 : BOOL;
		EditaciaMena_ENABLE : BOOL;
		EditaciaHesla_ENABLE : BOOL;
		EditaciaKarty_ENABLE : BOOL;
		TL_UlozUzivatela_ENABLE : BOOL;
		TlacitkoPrihlasenie_ENABLE : BOOL;
		Stav_ExistujuciUzivatel : BOOL;
		Stav_ChybajuceDataUzivatela : BOOL;
		StavyUsers_Index : USINT;
	END_STRUCT;
	ParametreUzivatelovTyp : 	STRUCT
		Meno : STRING[80];
		Heslo : STRING[80];
		CisloKarty : STRING[80];
		UrovenUzivatela : UINT;
	END_STRUCT;
END_TYPE
```

### UsersGlobal.var - Global variables
```iecst
VAR
	UsersVizu : UsersVizu_typ;
	MpRecipeXml_1 : MpRecipeXml := (0);
	MpRecipeRegPar_1 : MpRecipeRegPar := (0);
	Uzivatel : ARRAY[0..100] OF ParametreUzivatelovTyp;
	PrecitaneData_Panel1 : ARRAY[0..19] OF UDINT;
	PrecitaneData_Panel2 : ARRAY[0..19] OF UDINT;
	PrecitaneData_Panel3 : ARRAY[0..19] OF UDINT;
	PrecitaneData_Panel4 : ARRAY[0..19] OF UDINT;
	CisloPrihlasenejKarty_Panel1 : STRING[80];
	P1_UzivatelPrihlaseny : BOOL;
	P1_UrovenPrihlasenehoUzivatela : UINT; (*10 - operator, 20 - technik, 100 - administrátor*)
	P2_UzivatelPrihlaseny : BOOL;
	P2_UrovenPrihlasenehoUzivatela : UINT; (*10 - operator, 20 - technik, 100 - administrátor*)
	P34_UzivatelPrihlaseny : BOOL;
	P34_UrovenPrihlasenehoUzivatela : UINT; (*10 - operator, 20 - technik, 100 - administrátor*)
	Citacka1_AKTIVNA : BOOL;
	Citacka2_AKTIVNA : BOOL;
	Citacka3_AKTIVNA : BOOL;
END_VAR
```

### Program Logical/Uzivatelia/RFID_Prg (IEC)

#### RFID_Prg.st - Implementation code
```iecst
(********************************************************************
 * COPYRIGHT -- Bernecker + Rainer
 ********************************************************************
 * Program: RFID_Prg
 * File: RFID_Prg.st
 * Author: borsm
 * Created: December 23, 2015
 ********************************************************************
 * Implementation of program RFID_Prg
 ********************************************************************)

PROGRAM _INIT

    doinit:=1;

END_PROGRAM

PROGRAM _CYCLIC

	//Reset čitačiek RFID//
    IF NOT CasResetovaniaCitaciekRFID.Q THEN
        CasResetovaniaCitaciekRFID.IN:= TRUE;
    ELSIF CasResetovaniaCitaciekRFID.Q THEN
        doinit:= TRUE;
        CasResetovaniaCitaciekRFID.IN:= FALSE;
    END_IF

    CasResetovaniaCitaciekRFID.PT:= T#5m;
    CasResetovaniaCitaciekRFID();

(* find the Transponder, and give the Device ID back, this FuB works only for USB interface Transponder,

IF you use a serial interface transponder, please give the adress OF Interface ID directly TO the ident OF all FuBs *)

//Hladanie RFID čitačky//
    IF doinit THEN
        InitDone:= FALSE;
        doRead:= FALSE;
        TP_Init_0.Enable := TRUE;
        IF TP_Init_0.Done THEN
            PoruchaVyhladaniaCitaciek:= FALSE;
            DeviceID1 := TP_Init_0.Ident[2]; //Panel č.1
            DeviceID2 := TP_Init_0.Ident[1]; //Panel č.2
            DeviceID3 := TP_Init_0.Ident[0]; //Panel č.3
            TP_Init_0.Enable := FALSE;
            poc := poc + 1;
            IF poc	>= 3 THEN
                InitDone:= TRUE;
                doRead := TRUE;
                doinit:= FALSE;
                poc := 0;
            END_IF
        ELSIF TP_Init_0.Error THEN
            PoruchaVyhladaniaCitaciek:= TRUE;
            TP_Init_0.Enable := FALSE;
            doRead:= FALSE;
            doinit := FALSE;
        END_IF
    END_IF

    (* Čítanie z čítačky *)

    IF doRead AND InitDone AND NOT InitError THEN

        //Panel 1//
        TP_Read_1.Ident := DeviceID1;
        TP_Read_1.Enable := TRUE;
        IF TP_Read_1.Done THEN
            strcpy(ADR(READDATA_Citacka1),TP_Read_1.Data);
            TP_Read_1.Enable := FALSE;
        ELSIF TP_Read_1.Error THEN
            memset(ADR(READDATA_Citacka1),0,SIZEOF(READDATA_Citacka1));
            TP_Read_1.Enable := FALSE;
        END_IF

        //Panel 2//
        TP_Read_2.Ident := DeviceID2;
        TP_Read_2.Enable := TRUE;
        IF TP_Read_2.Done THEN
            strcpy(ADR(READDATA_Citacka2),TP_Read_2.Data);
            TP_Read_2.Enable := FALSE;
        ELSIF TP_Read_2.Error THEN
            memset(ADR(READDATA_Citacka2),0,SIZEOF(READDATA_Citacka2));
            TP_Read_2.Enable := FALSE;
        END_IF

        //Panel 3//
        TP_Read_3.Ident := DeviceID3;
        TP_Read_3.Enable := TRUE;
        IF TP_Read_3.Done THEN
           strcpy(ADR(READDATA_Citacka3),TP_Read_3.Data);
           TP_Read_3.Enable := FALSE;
        ELSIF TP_Read_3.Error THEN
           memset(ADR(READDATA_Citacka3),0,SIZEOF(READDATA_Citacka3));
           TP_Read_3.Enable := FALSE;
        END_IF

    ELSE
        TP_Read_1.Enable := FALSE;
        TP_Read_2.Enable := FALSE;
        TP_Read_3.Enable := FALSE;
        memset(ADR(READDATA_Citacka1),0,SIZEOF(READDATA_Citacka1));
        memset(ADR(READDATA_Citacka2),0,SIZEOF(READDATA_Citacka2));
        memset(ADR(READDATA_Citacka3),0,SIZEOF(READDATA_Citacka3));
    END_IF

    (* call FuBs *)
    TP_Init_0();
    TP_Read_1();
    TP_Read_2();
    TP_Read_3();

    //Zistenie či je priložená karta na čitačke 1//
    IF READDATA_Citacka1[2] = 0
        AND READDATA_Citacka1[3] = 0
        AND READDATA_Citacka1[4] = 0
        AND READDATA_Citacka1[5] = 0
        AND READDATA_Citacka1[6] = 0
        AND READDATA_Citacka1[7] = 0
        AND READDATA_Citacka1[8] = 0
        AND READDATA_Citacka1[9] = 0 THEN
        Citacka1_AKTIVNA:= FALSE;
    ELSE
        Citacka1_AKTIVNA:= TRUE;
    END_IF

    //Zistenie či je priložená karta na čitačke 2//
    IF READDATA_Citacka2[2] = 0
        AND READDATA_Citacka2[3] = 0
        AND READDATA_Citacka2[4] = 0
        AND READDATA_Citacka2[5] = 0
        AND READDATA_Citacka2[6] = 0
        AND READDATA_Citacka2[7] = 0
        AND READDATA_Citacka2[8] = 0
        AND READDATA_Citacka2[9] = 0 THEN
        Citacka2_AKTIVNA:= FALSE;
    ELSE
        Citacka2_AKTIVNA:= TRUE;
    END_IF

    //Zistenie či je priložená karta na čitačke 3//
    IF READDATA_Citacka3[2] = 0
        AND READDATA_Citacka3[3] = 0
        AND READDATA_Citacka3[4] = 0
        AND READDATA_Citacka3[5] = 0
        AND READDATA_Citacka3[6] = 0
        AND READDATA_Citacka3[7] = 0
        AND READDATA_Citacka3[8] = 0
        AND READDATA_Citacka3[9] = 0 THEN
        Citacka3_AKTIVNA:= FALSE;
    ELSE
        Citacka3_AKTIVNA:= TRUE;
    END_IF

    //Načítané kódy čitačiek//
    //Panel 1//
    IF P1_Vizu.TL_PrihlasovOperatora_AKTIVNE THEN  //Panel 1//
        IF Citacka1_AKTIVNA THEN
            PrecitaneData_Panel1[0]:= READDATA_Citacka1[3];
            PrecitaneData_Panel1[1]:= READDATA_Citacka1[2];
            PrecitaneData_Panel1[2]:= READDATA_Citacka1[5];
            PrecitaneData_Panel1[3]:= READDATA_Citacka1[4];
            PrecitaneData_Panel1[4]:= READDATA_Citacka1[7];
            PrecitaneData_Panel1[5]:= READDATA_Citacka1[6];
            PrecitaneData_Panel1[6]:= READDATA_Citacka1[9];
            PrecitaneData_Panel1[7]:= READDATA_Citacka1[8];
        ELSIF Citacka2_AKTIVNA THEN
            PrecitaneData_Panel1[0]:= READDATA_Citacka2[3];
            PrecitaneData_Panel1[1]:= READDATA_Citacka2[2];
            PrecitaneData_Panel1[2]:= READDATA_Citacka2[5];
            PrecitaneData_Panel1[3]:= READDATA_Citacka2[4];
            PrecitaneData_Panel1[4]:= READDATA_Citacka2[7];
            PrecitaneData_Panel1[5]:= READDATA_Citacka2[6];
            PrecitaneData_Panel1[6]:= READDATA_Citacka2[9];
            PrecitaneData_Panel1[7]:= READDATA_Citacka2[8];
        ELSIF Citacka3_AKTIVNA THEN
            PrecitaneData_Panel1[0]:= READDATA_Citacka3[3];
            PrecitaneData_Panel1[1]:= READDATA_Citacka3[2];
            PrecitaneData_Panel1[2]:= READDATA_Citacka3[5];
            PrecitaneData_Panel1[3]:= READDATA_Citacka3[4];
            PrecitaneData_Panel1[4]:= READDATA_Citacka3[7];
            PrecitaneData_Panel1[5]:= READDATA_Citacka3[6];
            PrecitaneData_Panel1[6]:= READDATA_Citacka3[9];
            PrecitaneData_Panel1[7]:= READDATA_Citacka3[8];
        END_IF
    ELSIF P2_Vizu.TL_PrihlasovOperatora_AKTIVNE THEN  //Panel 2//
        IF Citacka1_AKTIVNA THEN
            PrecitaneData_Panel2[0]:= READDATA_Citacka1[3];
            PrecitaneData_Panel2[1]:= READDATA_Citacka1[2];
            PrecitaneData_Panel2[2]:= READDATA_Citacka1[5];
            PrecitaneData_Panel2[3]:= READDATA_Citacka1[4];
            PrecitaneData_Panel2[4]:= READDATA_Citacka1[7];
            PrecitaneData_Panel2[5]:= READDATA_Citacka1[6];
            PrecitaneData_Panel2[6]:= READDATA_Citacka1[9];
            PrecitaneData_Panel2[7]:= READDATA_Citacka1[8];
        ELSIF Citacka2_AKTIVNA THEN
            PrecitaneData_Panel2[0]:= READDATA_Citacka2[3];
            PrecitaneData_Panel2[1]:= READDATA_Citacka2[2];
            PrecitaneData_Panel2[2]:= READDATA_Citacka2[5];
            PrecitaneData_Panel2[3]:= READDATA_Citacka2[4];
            PrecitaneData_Panel2[4]:= READDATA_Citacka2[7];
            PrecitaneData_Panel2[5]:= READDATA_Citacka2[6];
            PrecitaneData_Panel2[6]:= READDATA_Citacka2[9];
            PrecitaneData_Panel2[7]:= READDATA_Citacka2[8];
        ELSIF Citacka3_AKTIVNA THEN
            PrecitaneData_Panel2[0]:= READDATA_Citacka3[3];
            PrecitaneData_Panel2[1]:= READDATA_Citacka3[2];
            PrecitaneData_Panel2[2]:= READDATA_Citacka3[5];
            PrecitaneData_Panel2[3]:= READDATA_Citacka3[4];
            PrecitaneData_Panel2[4]:= READDATA_Citacka3[7];
            PrecitaneData_Panel2[5]:= READDATA_Citacka3[6];
            PrecitaneData_Panel2[6]:= READDATA_Citacka3[9];
            PrecitaneData_Panel2[7]:= READDATA_Citacka3[8];
        END_IF
    ELSIF P34_Vizu.TL_PrihlasovOperatora_AKTIVNE THEN  //Panel 3//
        IF Citacka1_AKTIVNA THEN
            PrecitaneData_Panel3[0]:= READDATA_Citacka1[3];
            PrecitaneData_Panel3[1]:= READDATA_Citacka1[2];
            PrecitaneData_Panel3[2]:= READDATA_Citacka1[5];
            PrecitaneData_Panel3[3]:= READDATA_Citacka1[4];
            PrecitaneData_Panel3[4]:= READDATA_Citacka1[7];
            PrecitaneData_Panel3[5]:= READDATA_Citacka1[6];
            PrecitaneData_Panel3[6]:= READDATA_Citacka1[9];
            PrecitaneData_Panel3[7]:= READDATA_Citacka1[8];
        ELSIF Citacka2_AKTIVNA THEN
            PrecitaneData_Panel3[0]:= READDATA_Citacka2[3];
            PrecitaneData_Panel3[1]:= READDATA_Citacka2[2];
            PrecitaneData_Panel3[2]:= READDATA_Citacka2[5];
            PrecitaneData_Panel3[3]:= READDATA_Citacka2[4];
            PrecitaneData_Panel3[4]:= READDATA_Citacka2[7];
            PrecitaneData_Panel3[5]:= READDATA_Citacka2[6];
            PrecitaneData_Panel3[6]:= READDATA_Citacka2[9];
            PrecitaneData_Panel3[7]:= READDATA_Citacka2[8];
        ELSIF Citacka3_AKTIVNA THEN
            PrecitaneData_Panel3[0]:= READDATA_Citacka3[3];
            PrecitaneData_Panel3[1]:= READDATA_Citacka3[2];
            PrecitaneData_Panel3[2]:= READDATA_Citacka3[5];
            PrecitaneData_Panel3[3]:= READDATA_Citacka3[4];
            PrecitaneData_Panel3[4]:= READDATA_Citacka3[7];
            PrecitaneData_Panel3[5]:= READDATA_Citacka3[6];
            PrecitaneData_Panel3[6]:= READDATA_Citacka3[9];
            PrecitaneData_Panel3[7]:= READDATA_Citacka3[8];
        END_IF
    ELSE
        PrecitaneData_Panel1[0]:= 0;
        PrecitaneData_Panel1[1]:= 0;
        PrecitaneData_Panel1[2]:= 0;
        PrecitaneData_Panel1[3]:= 0;
        PrecitaneData_Panel1[4]:= 0;
        PrecitaneData_Panel1[5]:= 0;
        PrecitaneData_Panel1[6]:= 0;
        PrecitaneData_Panel1[7]:= 0;

        PrecitaneData_Panel2[0]:= 0;
        PrecitaneData_Panel2[1]:= 0;
        PrecitaneData_Panel2[2]:= 0;
        PrecitaneData_Panel2[3]:= 0;
        PrecitaneData_Panel2[4]:= 0;
        PrecitaneData_Panel2[5]:= 0;
        PrecitaneData_Panel2[6]:= 0;
        PrecitaneData_Panel2[7]:= 0;

        PrecitaneData_Panel3[0]:= 0;
        PrecitaneData_Panel3[1]:= 0;
        PrecitaneData_Panel3[2]:= 0;
        PrecitaneData_Panel3[3]:= 0;
        PrecitaneData_Panel3[4]:= 0;
        PrecitaneData_Panel3[5]:= 0;
        PrecitaneData_Panel3[6]:= 0;
        PrecitaneData_Panel3[7]:= 0;
    END_IF

END_PROGRAM
```

#### RFID_Prg.var - Local variables
```iecst
(********************************************************************
 * COPYRIGHT -- Bernecker + Rainer
 ********************************************************************
 * Program: RFID_Prg
 * File: RFID_Prg.var
 * Author: borsm
 * Created: December 23, 2015
 ********************************************************************
 * Local variables of program RFID_Prg
 ********************************************************************)
VAR
	TP_Read_4 : TP_Read;
	TP_Read_1 : TP_Read;
	TP_Read_2 : TP_Read;
	TP_Read_3 : TP_Read;
	DeviceID1 : UDINT;
	DeviceID2 : UDINT;
	DeviceID3 : UDINT;
	DeviceID4 : UDINT;
	READDATA_Citacka1 : ARRAY[0..19] OF USINT;
	READDATA_Citacka2 : ARRAY[0..19] OF USINT;
	READDATA_Citacka3 : ARRAY[0..19] OF USINT;
	READDATA_Citacka4 : ARRAY[0..19] OF USINT;
	TP_Write_0 : TP_Write;
	WRITEDATA : STRING[8];
	ReadDone_Panel1 : BOOL;
	ReadDone_Panel2 : BOOL;
	ReadDone_Panel3 : BOOL;
	ReadError_Panel1 : BOOL;
	ReadError_Panel2 : BOOL;
	ReadError_Panel3 : BOOL;
	ReadErrorID_Panel1 : UDINT;
	ReadErrorID_Panel2 : UDINT;
	ReadErrorID_Panel3 : UDINT;
	doRead : BOOL;
	doWrite : BOOL;
	WriteDone : BOOL;
	WriteError : BOOL;
	WriteErrorID : UDINT;
	TP_Init_0 : TP_Init;
	TP_OnOff_0 : TP_OnOff;
	TP_Crc_0 : TP_Crc;
	TP_Lock_0 : TP_Lock;
	TP_Info_0 : TP_Info;
	TP_PWProtect_0 : TP_PWProtect;
	TP_Unlock_0 : TP_Unlock;
	doPassword : BOOL;
	PasswordErrorID : UDINT;
	PasswordError : BOOL;
	PasswordDone : BOOL;
	passwordin : STRING[8];
	doUnlock : BOOL;
	UnlockErrorID : UDINT;
	UnlockError : BOOL;
	UnlockDone : BOOL;
	password : STRING[8];
	doLock : BOOL;
	LockErrorID : UDINT;
	LockError : BOOL;
	LockDone : BOOL;
	doCrc : BOOL;
	CrcErrorID : UDINT;
	CrcError : BOOL;
	CrcDone : BOOL;
	doInfo : BOOL;
	InfoErrorID : UDINT;
	InfoError : BOOL;
	InfoDone : BOOL;
	sl : ARRAY[0..1] OF USINT;
	KEYTYPE : ARRAY[0..3] OF USINT;
	Type : ARRAY[0..30] OF USINT;
	ID : ARRAY[0..9] OF USINT;
	doOnOff : BOOL;
	OnOffDone : BOOL;
	OnOffErrorID : UDINT;
	OnOffError : BOOL;
	InitDone : BOOL;
	InitErrorID : UDINT;
	InitError : BOOL;
	poc : USINT;
	step : INT;
	doinit : BOOL;
	CasResetovaniaCitaciekRFID : TON;
	PoruchaVyhladaniaCitaciek : BOOL;
	TEST : BOOL;
	a : USINT;
	b : USINT;
	c : USINT;
END_VAR
```

### Program Logical/Uzivatelia/Users_Main (IEC)

#### Main.st - Init, cyclic, exit code
```iecst
PROGRAM _INIT
	MpRecipeXml_1.Load:= TRUE;

END_PROGRAM

PROGRAM _CYCLIC

	//Volanie funkcie SequenceControl//
	SequenceControl(SC:= SC_Uzivatelia);

	//Načítanie receptur z pamäte//
	IF MpRecipeXml_1.Load AND (MpRecipeXml_1.CommandDone OR MpRecipeXml_1.Error) THEN
		MpRecipeXml_1.Load:= FALSE;
	END_IF

	//Konfigurácia receptur//
	MpRecipeXml_1.MpLink:= ADR(gUserXml);  //takto sa menuje mapp komponenta v configurating view//
	MpRecipeXml_1.Enable:= TRUE;
	MpRecipeXml_1.Category:= ADR('UZIVATELIA');
	MpRecipeXml_1.Category:= ADR(strCategory);
	MpRecipeXml_1.DeviceName:= ADR('HDD_Users');  //Názov media, kde sa budú receptury ukladat//
	MpRecipeXml_1.FileName:= ADR('UlozeniUzivatelia'); //Názov súboru do ktorého sa receptúry uložia//
	MpRecipeXml_1();

	MpRecipeRegPar_1.MpLink:= ADR(gUserXml);
	MpRecipeRegPar_1.Enable:= TRUE;
	MpRecipeRegPar_1.Category:= ADR('UZIVATELIA');
	MpRecipeRegPar_1.PVName:= ADR('Uzivatel'); //Názov premenné, kde je vytvorená štruktura dat pre receptury//
	MpRecipeRegPar_1();

    //Zamknutie tlačítka Uloženie uživatelov//
    IF UsersVizu.Edit_MenoUzivatela = '' THEN
        UsersVizu.TL_UlozUzivatela_ENABLE:= FALSE;
    ELSIF UsersVizu.Edit_CisloKarty = '' THEN
        UsersVizu.TL_UlozUzivatela_ENABLE:= FALSE;
    ELSE
        UsersVizu.TL_UlozUzivatela_ENABLE:= TRUE;
   END_IF

    //Zobrazenie zoznamu uživatelov//

    FOR a:= 0 TO 100 BY 1 DO
        ListBoxPole_Sprava[a]:= '{"value":"';
        ListBox_Value[a]:= UINT_TO_STRING(a);
        brsstrcat(ADR(ListBoxPole_Sprava[a]), ADR(ListBox_Value[a]));
        brsstrcat(ADR(ListBoxPole_Sprava[a]), ADR('","text":"'));
        brsstrcat(ADR(ListBoxPole_Sprava[a]), ADR(Uzivatel[a].Meno));
        brsstrcat(ADR(ListBoxPole_Sprava[a]), ADR('"}'));
        IF Uzivatel[a].Meno = '' THEN
            UsersVizu.ZoznamUzivatelov[a]:= '';
        ELSE
            UsersVizu.ZoznamUzivatelov[a]:= ListBoxPole_Sprava[a];
        END_IF
    END_FOR

    //Vyčítanie aktuálneho indexu text listu (hodnota string) a prevod do premennej UINT//
    e:= STRING_TO_UINT(UsersVizu.LB_IndexSTRING);

    //Načítanie čísla karty//
    IF P1_Vizu.TL_PrihlasovOperatora_AKTIVNE AND (Citacka1_AKTIVNA OR Citacka2_AKTIVNA OR Citacka3_AKTIVNA) THEN
        UsersVizu.Edit_CisloKarty:= CisloPrihlasenejKarty_Panel1;
    END_IF

    IF NOT P1_Vizu.TL_PrihlasovOperatora_AKTIVNE THEN
        UsersVizu.Edit_CisloKarty:= '';
    END_IF

    //***************************************Editácia databáze uzivatelov*********************************//
    CASE SC_Uzivatelia.Step OF

        0://Vynulovanie uživatela//
            SC_Uzivatelia.StepName:= '0 - Nulovanie';
            UsersVizu.UlozUzivatela:= FALSE;
            UsersVizu.VymazUzivatela:= FALSE;
            UsersVizu.NacitajUzivatela:= FALSE;

            MpRecipeXml_1.Save:= FALSE;
            i:= 0;
            c:= 0;
            d:= 0;
            IndexPrazdPole:= 0;
            SC_Uzivatelia.ResetStep:= TRUE;
            SC_Uzivatelia.Step:= 1;

        1://Rozhodnutie o činnosti//
            SC_Uzivatelia.StepName:= '1 - Rozhodnutie o cinnosti';
            IF UsersVizu.UlozUzivatela THEN
                SC_Uzivatelia.Step:= 10;
            ELSIF UsersVizu.NacitajUzivatela THEN
                SC_Uzivatelia.Step:= 20;
            ELSIF UsersVizu.VymazUzivatela THEN
                SC_Uzivatelia.Step:= 30;
            END_IF

        10://Kontrola zadaných udajov uzivatela//
            SC_Uzivatelia.StepName:= '10 - Kontrola zadanych udajov uzivatela';
            UsersVizu.StavyUsers_Index:= 9;
            IF UsersVizu.Edit_MenoUzivatela = '' OR UsersVizu.Edit_CisloKarty = '' THEN
                UsersVizu.StavyUsers_Index:= 13; //Zobrazenie stavov v textovom okne
                SC_Uzivatelia.ResetStep:= TRUE;
                SC_Uzivatelia.Step:= 0;
            ELSE
                SC_Uzivatelia.ResetStep:= TRUE;
                SC_Uzivatelia.Step:= 11;
            END_IF

        11://Kontrola mena už existujucich uzivatelov//
            SC_Uzivatelia.StepName:= '11 - Kontrola mena uz existujucich uzivatelov';
            IF Uzivatel[c].Meno = UsersVizu.Edit_MenoUzivatela THEN
                UsersVizu.StavyUsers_Index:= 2;
                SC_Uzivatelia.ResetStep:= TRUE;
                SC_Uzivatelia.Step:= 0;
            ELSE
                IF c < 100 THEN
                    c:= c + 1;
                ELSE
                    SC_Uzivatelia.ResetStep:= TRUE;
					SC_Uzivatelia.Step:= 12;
				END_IF
			END_IF

		12://Zistenie prázdneho pola pre uloženie receptury//
			SC_Uzivatelia.StepName:= '12 - Zistenie volneho pola';
			IF Uzivatel[d].Meno= '' THEN
				IndexPrazdPole:= d;
				SC_Uzivatelia.ResetStep:= TRUE;
				SC_Uzivatelia.Step:= 13;
			ELSE
				IF d < 100 THEN
					d:= d + 1;
				ELSE
					SC_Uzivatelia.ResetStep:= TRUE;
					SC_Uzivatelia.Step:= 0;
				END_IF
			END_IF

		13://Ulozenie uzivatela//
			SC_Uzivatelia.StepName:= '13 - Ulozenie uzivatela';
			Uzivatel[IndexPrazdPole].Meno:= UsersVizu.Edit_MenoUzivatela;
            Uzivatel[IndexPrazdPole].CisloKarty:= UsersVizu.Edit_CisloKarty;
            UrovenUzivatela:= STRING_TO_UINT(UsersVizu.Edit_UrovenUzivatela);
            Uzivatel[IndexPrazdPole].UrovenUzivatela:= UrovenUzivatela;
            MpRecipeXml_1.Save:= TRUE;
            IF MpRecipeXml_1.CommandDone THEN
                UsersVizu.StavyUsers_Index:= 1;
                UsersVizu.Edit_MenoUzivatela:= '';
                UsersVizu.Edit_CisloKarty:= '';
                SC_Uzivatelia.ResetStep:= TRUE;
                SC_Uzivatelia.Step:= 0;
		    END_IF

        20://Načítanie parametrov uživatela//
            SC_Uzivatelia.StepName:= '20 - Nacitanie parametrov uzivatela';
            UsersVizu.StavyUsers_Index:= 9;
            UsersVizu.Edit_MenoUzivatela:= Uzivatel[e].Meno;
            UsersVizu.Edit_HesloUzivatela:= Uzivatel[e].Heslo;
            UrovenUzivatela:= Uzivatel[e].UrovenUzivatela;
            UsersVizu.Edit_UrovenUzivatela:= UINT_TO_STRING(UrovenUzivatela);
            (*UsersVizu.Edit_CisloKarty:= Uzivatel[e].CisloKarty;*)
            UsersVizu.StavyUsers_Index:= 3;
            SC_Uzivatelia.ResetStep:= TRUE;
            SC_Uzivatelia.Step:= 0;

        30://Vymazanie uživatela//
            SC_Uzivatelia.StepName:= '30 - Vymazanie uzivatela';
            UsersVizu.StavyUsers_Index:= 9;
            Uzivatel[e].Meno:= '';
            Uzivatel[e].Heslo:= '';
            Uzivatel[e].CisloKarty:= '';
            Uzivatel[e].UrovenUzivatela:= 0;
            MpRecipeXml_1.Save:= TRUE;
            IF MpRecipeXml_1.CommandDone THEN
                UsersVizu.StavyUsers_Index:= 4;
                SC_Uzivatelia.ResetStep:= TRUE;
                SC_Uzivatelia.Step:= 0;
            END_IF

    END_CASE

				END_PROGRAM

PROGRAM _EXIT
				(* Insert code here *)

				END_PROGRAM
```

#### Variables.var - Local variables
```iecst
VAR
	strCategory : STRING[80];
	MpRecipeUI_1 : MpRecipeUI;
	UISetup : MpRecipeUISetupType;
	UIConnect : MpRecipeUIConnectType := (0);
	i : UINT := 0;
	a : UINT;
	CasOdhlaseniaUzivatela : TON;
	ListBoxPole_Sprava : ARRAY[0..100] OF STRING[100];
	ListBox_Value : ARRAY[0..100] OF STRING[10];
	b : USINT;
	c : UINT;
	IndexPrazdPole : UINT;
	d : UINT;
	e : UINT;
	f : UINT;
	g : UINT;
	h : UINT;
	SC_Uzivatelia : SequenceControlTyp;
	UrovenUzivatela : UINT;
END_VAR
```

### Program Logical/Uzivatelia/Users_Panel1 (IEC)

#### Main.st - Init, cyclic, exit code
```iecst
PROGRAM _INIT

END_PROGRAM

PROGRAM _CYCLIC

    //Volanie funkcie SequenceControl//
    SequenceControl(SC:= SC_Uzivatelia);

    //************************************Konvertovanie kódu čitačky do stringu****************************************************//
    FOR i:= 0 TO 7 BY 1 DO
        brsstrcpy(ADR(PrecitaneDataSTRING[i]),ADR(PrecitaneData_Panel1[i]));
    END_FOR

    //Spajanie pola stringov do stringu//
    KodCitackySTRING:= PrecitaneDataSTRING[0];
    brsstrcat(ADR(KodCitackySTRING), ADR(PrecitaneDataSTRING[1]));
    brsstrcat(ADR(KodCitackySTRING), ADR(PrecitaneDataSTRING[2]));
    brsstrcat(ADR(KodCitackySTRING), ADR(PrecitaneDataSTRING[3]));
    brsstrcat(ADR(KodCitackySTRING), ADR(PrecitaneDataSTRING[4]));
    brsstrcat(ADR(KodCitackySTRING), ADR(PrecitaneDataSTRING[5]));
    brsstrcat(ADR(KodCitackySTRING), ADR(PrecitaneDataSTRING[6]));
    brsstrcat(ADR(KodCitackySTRING), ADR(PrecitaneDataSTRING[7]));

    IF KodCitackySTRING = '' THEN
        CisloPrihlasenejKarty_Panel1:= '';
    ELSE
        CisloPrihlasenejKarty_Panel1:= KodCitackySTRING;
    END_IF

    //**************************************************Kontrola či je karta priložená******************************************************//

    IF KodCitackySTRING <> '' THEN
        CasControlyKarty.IN:= TRUE;
    ELSE
        CasControlyKarty.IN:= FALSE;
    END_IF

    IF CasControlyKarty.Q THEN
        UsersVizu.KartaPrilozena_Panel1:= TRUE;
    ELSE
        UsersVizu.KartaPrilozena_Panel1:= FALSE;
    END_IF

    CasControlyKarty.PT:= T#1s;
    CasControlyKarty();

    //***************************************************Kontrola či je uživatel už prihlásený**********************************************//
    IF UsersVizu.MenoPrihlasenehoUzivatela_Panel1 = '' THEN
        P1_UzivatelPrihlaseny:= FALSE;
    ELSE
        P1_UzivatelPrihlaseny:= TRUE;
    END_IF
//    P1_UzivatelPrihlaseny:= TRUE;
//    P1_UrovenPrihlasenehoUzivatela:= 20;

    //Kontrola karty//

    IF KodCitackySTRING = '' THEN
        PrecitaneCisloKarty:= '';
    ELSE
        PrecitaneCisloKarty:= KodCitackySTRING;
    END_IF

    CASE SC_Uzivatelia.Step OF

        0://Nulovanie//
            SC_Uzivatelia.StepName:= '0 - Nulovanie';
            UsersVizu.OdhlasUzivatela_Panel1:= FALSE;
            a:= 0;
            SC_Uzivatelia.ResetStep:= TRUE;
            SC_Uzivatelia.Step:= 1;

        1://Rozhodnutie o činnosti//
            SC_Uzivatelia.StepName:= '1 - Rozhodnutie o cinnosti';
            IF UsersVizu.KartaPrilozena_Panel1 AND P1_Vizu.ActualPage <> 'PageUsers' THEN
                SC_Uzivatelia.ResetStep:= TRUE;
                SC_Uzivatelia.Step:= 10;
            ELSIF UsersVizu.OdhlasUzivatela_Panel1 THEN
                SC_Uzivatelia.ResetStep:= TRUE;
                SC_Uzivatelia.Step:= 20;
            END_IF

        10://Kontrola udajov karty//
            SC_Uzivatelia.StepName:= '10 - Kontrola udajov karty';
            SC_Uzivatelia.IdleTime.PT:= T#2s;
            SC_Uzivatelia.AlarmTime.PT:= T#2s;

            IF NOT P1_UzivatelPrihlaseny THEN
                IF PrecitaneCisloKarty <> '' THEN
                    SC_Uzivatelia.ResetStep:= TRUE;
                    SC_Uzivatelia.Step:= 13;
                ELSE
                    SC_Uzivatelia.ResetStep:= TRUE;
                    SC_Uzivatelia.Step:= 100;
                END_IF
            ELSE
                SC_Uzivatelia.ResetStep:= TRUE;
                SC_Uzivatelia.Step:= 100;
            END_IF

        13://Hladanie prihlaseného uživatela v zoznamoch//
            SC_Uzivatelia.StepName:= '13 - Hladanie prihlaseneho uzivatela';
            SC_Uzivatelia.IdleTime.PT:= T#2s;
            SC_Uzivatelia.AlarmTime.PT:= T#2s;

            IF Uzivatel[a].CisloKarty = PrecitaneCisloKarty THEN
                UsersVizu.MenoPrihlasenehoUzivatela_Panel1:= Uzivatel[a].Meno;
                UsersVizu.CisloPrihlasenejKarty_Panel1:= Uzivatel[a].CisloKarty;
                P1_UrovenPrihlasenehoUzivatela:= Uzivatel[a].UrovenUzivatela;
                SC_Uzivatelia.ResetStep:= TRUE;
                SC_Uzivatelia.Step:= 100;
            ELSE
                IF a < 100 THEN
                    a:= a + 1;
                ELSE
                    SC_Uzivatelia.ResetStep:= TRUE;
                    SC_Uzivatelia.Step:= 15;
                END_IF
            END_IF

        15://Priradenie čísla karty//
            SC_Uzivatelia.StepName:= '15 - Priradenie cisla karty';
            SC_Uzivatelia.IdleTime.PT:= T#2s;
            SC_Uzivatelia.AlarmTime.PT:= T#2s;

            UsersVizu.MenoPrihlasenehoUzivatela_Panel1:= 'Operator';
            UsersVizu.CisloPrihlasenejKarty_Panel1:= PrecitaneCisloKarty;
            SC_Uzivatelia.ResetStep:= TRUE;
            SC_Uzivatelia.Step:= 100;

        20://Odhlásenie uživatela//
            SC_Uzivatelia.StepName:= '20 - Odhlasenie uzivatela';
            SC_Uzivatelia.IdleTime.PT:= T#2s;
            SC_Uzivatelia.AlarmTime.PT:= T#2s;

            UsersVizu.MenoPrihlasenehoUzivatela_Panel1:= '';
            UsersVizu.CisloPrihlasenejKarty_Panel1:= '';
            P1_UrovenPrihlasenehoUzivatela:= 0;
            SC_Uzivatelia.ResetStep:= TRUE;
            SC_Uzivatelia.Step:= 100;

        100://Čakam na odobratie karty//
            SC_Uzivatelia.StepName:= '110 - Cakanie na odobratie karty';
            SC_Uzivatelia.IdleTime.PT:= T#1s;
            SC_Uzivatelia.AlarmTime.PT:= T#2s;

            SC_Uzivatelia.IdleTime.IN:= NOT UsersVizu.KartaPrilozena_Panel1;

            IF SC_Uzivatelia.IdleTime.Q THEN
                SC_Uzivatelia.ResetStep:= TRUE;
                SC_Uzivatelia.Step:= 0;
            END_IF

    END_CASE

END_PROGRAM

PROGRAM _EXIT
	(* Insert code here *)

END_PROGRAM
```

#### Variables.var - Local variables
```iecst
VAR
	i : USINT;
	PrecitaneDataSTRING : ARRAY[0..7] OF STRING[1] := [8('')];
	KodCitackySTRING : STRING[80];
	CasControlyKarty : TON;
	SC_Uzivatelia : SequenceControlTyp;
	PrecitaneCisloKarty : STRING[80];
	a : USINT;
END_VAR
```

### Program Logical/Uzivatelia/Users_Panel2 (IEC)

#### Main.st - Init, cyclic, exit code
```iecst
PROGRAM _INIT

END_PROGRAM

PROGRAM _CYCLIC

    //Volanie funkcie SequenceControl//
    SequenceControl(SC:= SC_Uzivatelia);

    //************************************Konvertovanie kódu čitačky do stringu****************************************************//
    FOR i:= 0 TO 7 BY 1 DO
        brsstrcpy(ADR(PrecitaneDataSTRING[i]),ADR(PrecitaneData_Panel2[i]));
    END_FOR

    //Spajanie pola stringov do stringu//
    KodCitackySTRING:= PrecitaneDataSTRING[0];
    brsstrcat(ADR(KodCitackySTRING), ADR(PrecitaneDataSTRING[1]));
    brsstrcat(ADR(KodCitackySTRING), ADR(PrecitaneDataSTRING[2]));
    brsstrcat(ADR(KodCitackySTRING), ADR(PrecitaneDataSTRING[3]));
    brsstrcat(ADR(KodCitackySTRING), ADR(PrecitaneDataSTRING[4]));
    brsstrcat(ADR(KodCitackySTRING), ADR(PrecitaneDataSTRING[5]));
    brsstrcat(ADR(KodCitackySTRING), ADR(PrecitaneDataSTRING[6]));
    brsstrcat(ADR(KodCitackySTRING), ADR(PrecitaneDataSTRING[7]));

    //**************************************************Kontrola či je karta priložená******************************************************//

    IF KodCitackySTRING <> '' THEN
        CasControlyKarty.IN:= TRUE;
    ELSE
        CasControlyKarty.IN:= FALSE;
    END_IF

    IF CasControlyKarty.Q THEN
        UsersVizu.KartaPrilozena_Panel2:= TRUE;
    ELSE
        UsersVizu.KartaPrilozena_Panel2:= FALSE;
    END_IF

    CasControlyKarty.PT:= T#1s;
    CasControlyKarty();

    //***************************************************Kontrola či je uživatel už prihlásený**********************************************//
    IF UsersVizu.MenoPrihlasenehoUzivatela_Panel2 = '' THEN
        P2_UzivatelPrihlaseny:= FALSE;
    ELSE
        P2_UzivatelPrihlaseny:= TRUE;
    END_IF

//    P2_UzivatelPrihlaseny:= TRUE;
//    P2_UrovenPrihlasenehoUzivatela:= 20;

    //Kontrola karty//

    IF KodCitackySTRING = '' THEN
        PrecitaneCisloKarty:= '';
    ELSE
        PrecitaneCisloKarty:= KodCitackySTRING;
    END_IF

    CASE SC_Uzivatelia.Step OF

        0://Nulovanie//
            SC_Uzivatelia.StepName:= '0 - Nulovanie';
            UsersVizu.OdhlasUzivatela_Panel2:= FALSE;
            a:= 0;
            SC_Uzivatelia.ResetStep:= TRUE;
            SC_Uzivatelia.Step:= 1;

        1://Rozhodnutie o činnosti//
            SC_Uzivatelia.StepName:= '1 - Rozhodnutie o cinnosti';
            IF UsersVizu.KartaPrilozena_Panel2 THEN
                SC_Uzivatelia.ResetStep:= TRUE;
                SC_Uzivatelia.Step:= 10;
            ELSIF UsersVizu.OdhlasUzivatela_Panel2 THEN
                SC_Uzivatelia.ResetStep:= TRUE;
                SC_Uzivatelia.Step:= 20;
            END_IF

        10://Kontrola udajov karty//
            SC_Uzivatelia.StepName:= '10 - Kontrola udajov karty';
            SC_Uzivatelia.IdleTime.PT:= T#2s;
            SC_Uzivatelia.AlarmTime.PT:= T#2s;

            IF NOT P2_UzivatelPrihlaseny THEN
                IF PrecitaneCisloKarty <> '' THEN
                    SC_Uzivatelia.ResetStep:= TRUE;
                    SC_Uzivatelia.Step:= 13;
                ELSE
                    SC_Uzivatelia.ResetStep:= TRUE;
                    SC_Uzivatelia.Step:= 100;
                END_IF
            ELSE
                SC_Uzivatelia.ResetStep:= TRUE;
                SC_Uzivatelia.Step:= 100;
            END_IF

        13://Hladanie prihlaseného uživatela v zoznamoch//
            SC_Uzivatelia.StepName:= '13 - Hladanie prihlaseneho uzivatela';
            SC_Uzivatelia.IdleTime.PT:= T#2s;
            SC_Uzivatelia.AlarmTime.PT:= T#2s;

            IF Uzivatel[a].CisloKarty = PrecitaneCisloKarty THEN
                UsersVizu.MenoPrihlasenehoUzivatela_Panel2:= Uzivatel[a].Meno;
                UsersVizu.CisloPrihlasenejKarty_Panel2:= Uzivatel[a].CisloKarty;
                P2_UrovenPrihlasenehoUzivatela:= Uzivatel[a].UrovenUzivatela;
                SC_Uzivatelia.ResetStep:= TRUE;
                SC_Uzivatelia.Step:= 100;
            ELSE
                IF a < 100 THEN
                    a:= a + 1;
                ELSE
                    SC_Uzivatelia.ResetStep:= TRUE;
                    SC_Uzivatelia.Step:= 15;
                END_IF
            END_IF

        15://Priradenie čísla karty//
            SC_Uzivatelia.StepName:= '15 - Priradenie cisla karty';
            SC_Uzivatelia.IdleTime.PT:= T#2s;
            SC_Uzivatelia.AlarmTime.PT:= T#2s;

            UsersVizu.MenoPrihlasenehoUzivatela_Panel2:= 'Operator';
            UsersVizu.CisloPrihlasenejKarty_Panel2:= PrecitaneCisloKarty;
            SC_Uzivatelia.ResetStep:= TRUE;
            SC_Uzivatelia.Step:= 100;

        20://Odhlásenie uživatela//
            SC_Uzivatelia.StepName:= '20 - Odhlasenie uzivatela';
            SC_Uzivatelia.IdleTime.PT:= T#2s;
            SC_Uzivatelia.AlarmTime.PT:= T#2s;

            UsersVizu.MenoPrihlasenehoUzivatela_Panel2:= '';
            UsersVizu.CisloPrihlasenejKarty_Panel2:= '';
            P2_UrovenPrihlasenehoUzivatela:= 0;
            SC_Uzivatelia.ResetStep:= TRUE;
            SC_Uzivatelia.Step:= 100;

        100://Čakam na odobratie karty//
            SC_Uzivatelia.StepName:= '110 - Cakanie na odobratie karty';
            SC_Uzivatelia.IdleTime.PT:= T#1s;
            SC_Uzivatelia.AlarmTime.PT:= T#2s;

            SC_Uzivatelia.IdleTime.IN:= NOT UsersVizu.KartaPrilozena_Panel2;

            IF SC_Uzivatelia.IdleTime.Q THEN
                SC_Uzivatelia.ResetStep:= TRUE;
                SC_Uzivatelia.Step:= 0;
            END_IF

    END_CASE

END_PROGRAM

PROGRAM _EXIT
	(* Insert code here *)

END_PROGRAM
```

#### Variables.var - Local variables
```iecst
VAR
	i : USINT;
	PrecitaneDataSTRING : ARRAY[0..7] OF STRING[1] := [8('')];
	KodCitackySTRING : STRING[80];
	CasControlyKarty : TON;
	SC_Uzivatelia : SequenceControlTyp;
	PrecitaneCisloKarty : STRING[80];
	a : USINT;
END_VAR
```

### Program Logical/Uzivatelia/Users_Panel3 (IEC)

#### Main.st - Init, cyclic, exit code
```iecst
PROGRAM _INIT

END_PROGRAM

PROGRAM _CYCLIC

    //Volanie funkcie SequenceControl//
    SequenceControl(SC:= SC_Uzivatelia);

      //************************************Konvertovanie kódu čitačky do stringu****************************************************//
    FOR i:= 0 TO 7 BY 1 DO
        brsstrcpy(ADR(PrecitaneDataSTRING[i]),ADR(PrecitaneData_Panel3[i]));
    END_FOR

    //Spajanie pola stringov do stringu//
    KodCitackySTRING:= PrecitaneDataSTRING[0];
    brsstrcat(ADR(KodCitackySTRING), ADR(PrecitaneDataSTRING[1]));
    brsstrcat(ADR(KodCitackySTRING), ADR(PrecitaneDataSTRING[2]));
    brsstrcat(ADR(KodCitackySTRING), ADR(PrecitaneDataSTRING[3]));
    brsstrcat(ADR(KodCitackySTRING), ADR(PrecitaneDataSTRING[4]));
    brsstrcat(ADR(KodCitackySTRING), ADR(PrecitaneDataSTRING[5]));
    brsstrcat(ADR(KodCitackySTRING), ADR(PrecitaneDataSTRING[6]));
    brsstrcat(ADR(KodCitackySTRING), ADR(PrecitaneDataSTRING[7]));

    //**************************************************Kontrola či je karta priložená******************************************************//

    IF KodCitackySTRING <> '' THEN
        CasControlyKarty.IN:= TRUE;
    ELSE
        CasControlyKarty.IN:= FALSE;
    END_IF

    IF CasControlyKarty.Q THEN
        UsersVizu.KartaPrilozena_Panel3:= TRUE;
    ELSE
        UsersVizu.KartaPrilozena_Panel3:= FALSE;
    END_IF

    CasControlyKarty.PT:= T#1s;
    CasControlyKarty();

    //***************************************************Kontrola či je uživatel už prihlásený**********************************************//
    IF UsersVizu.MenoPrihlasenehoUzivatela_Panel3 = '' THEN
        P34_UzivatelPrihlaseny:= FALSE;
    ELSE
        P34_UzivatelPrihlaseny:= TRUE;
    END_IF

//    P34_UzivatelPrihlaseny:= TRUE;
//    P34_UrovenPrihlasenehoUzivatela:= 20;

    //Kontrola karty//

    IF KodCitackySTRING = '' THEN
        PrecitaneCisloKarty:= '';
    ELSE
        PrecitaneCisloKarty:= KodCitackySTRING;
    END_IF

    CASE SC_Uzivatelia.Step OF

        0://Nulovanie//
            SC_Uzivatelia.StepName:= '0 - Nulovanie';
            UsersVizu.OdhlasUzivatela_Panel3:= FALSE;
            a:= 0;
            SC_Uzivatelia.ResetStep:= TRUE;
            SC_Uzivatelia.Step:= 1;

        1://Rozhodnutie o činnosti//
            SC_Uzivatelia.StepName:= '1 - Rozhodnutie o cinnosti';
            IF UsersVizu.KartaPrilozena_Panel3 THEN
                SC_Uzivatelia.ResetStep:= TRUE;
                SC_Uzivatelia.Step:= 10;
            ELSIF UsersVizu.OdhlasUzivatela_Panel3 THEN
                SC_Uzivatelia.ResetStep:= TRUE;
                SC_Uzivatelia.Step:= 20;
            END_IF

        10://Kontrola udajov karty//
            SC_Uzivatelia.StepName:= '10 - Kontrola udajov karty';
            SC_Uzivatelia.IdleTime.PT:= T#2s;
            SC_Uzivatelia.AlarmTime.PT:= T#2s;

            IF NOT P34_UzivatelPrihlaseny THEN
                IF PrecitaneCisloKarty <> '' THEN
                    SC_Uzivatelia.ResetStep:= TRUE;
                    SC_Uzivatelia.Step:= 13;
                ELSE
                    SC_Uzivatelia.ResetStep:= TRUE;
                    SC_Uzivatelia.Step:= 100;
                END_IF
            ELSE
                SC_Uzivatelia.ResetStep:= TRUE;
                SC_Uzivatelia.Step:= 100;
            END_IF

        13://Hladanie prihlaseného uživatela v zoznamoch//
            SC_Uzivatelia.StepName:= '13 - Hladanie prihlaseneho uzivatela';
            SC_Uzivatelia.IdleTime.PT:= T#2s;
            SC_Uzivatelia.AlarmTime.PT:= T#2s;

            IF Uzivatel[a].CisloKarty = PrecitaneCisloKarty THEN
                UsersVizu.MenoPrihlasenehoUzivatela_Panel3:= Uzivatel[a].Meno;
                UsersVizu.CisloPrihlasenejKarty_Panel3:= Uzivatel[a].CisloKarty;
                P34_UrovenPrihlasenehoUzivatela:= Uzivatel[a].UrovenUzivatela;
                SC_Uzivatelia.ResetStep:= TRUE;
                SC_Uzivatelia.Step:= 100;
            ELSE
                IF a < 100 THEN
                    a:= a + 1;
                ELSE
                    SC_Uzivatelia.ResetStep:= TRUE;
                    SC_Uzivatelia.Step:= 15;
                END_IF
            END_IF

        15://Priradenie čísla karty//
            SC_Uzivatelia.StepName:= '15 - Priradenie cisla karty';
            SC_Uzivatelia.IdleTime.PT:= T#2s;
            SC_Uzivatelia.AlarmTime.PT:= T#2s;

            UsersVizu.MenoPrihlasenehoUzivatela_Panel3:= 'Operator';
            UsersVizu.CisloPrihlasenejKarty_Panel1:= PrecitaneCisloKarty;
            SC_Uzivatelia.ResetStep:= TRUE;
            SC_Uzivatelia.Step:= 100;

        20://Odhlásenie uživatela//
            SC_Uzivatelia.StepName:= '20 - Odhlasenie uzivatela';
            SC_Uzivatelia.IdleTime.PT:= T#2s;
            SC_Uzivatelia.AlarmTime.PT:= T#2s;

            UsersVizu.MenoPrihlasenehoUzivatela_Panel3:= '';
            UsersVizu.CisloPrihlasenejKarty_Panel3:= '';
            P34_UrovenPrihlasenehoUzivatela:= 0;
            SC_Uzivatelia.ResetStep:= TRUE;
            SC_Uzivatelia.Step:= 100;

        100://Čakam na odobratie karty//
            SC_Uzivatelia.StepName:= '110 - Cakanie na odobratie karty';
            SC_Uzivatelia.IdleTime.PT:= T#1s;
            SC_Uzivatelia.AlarmTime.PT:= T#2s;

            SC_Uzivatelia.IdleTime.IN:= NOT UsersVizu.KartaPrilozena_Panel3;

            IF SC_Uzivatelia.IdleTime.Q THEN
                SC_Uzivatelia.ResetStep:= TRUE;
                SC_Uzivatelia.Step:= 0;
            END_IF

    END_CASE

END_PROGRAM

PROGRAM _EXIT
	(* Insert code here *)

END_PROGRAM
```

#### Variables.var - Local variables
```iecst
VAR
	i : USINT;
	PrecitaneDataSTRING : ARRAY[0..7] OF STRING[1] := [8('')];
	KodCitackySTRING : STRING[80];
	CasControlyKarty : TON;
	SC_Uzivatelia : SequenceControlTyp;
	PrecitaneCisloKarty : STRING[80];
	a : USINT;
END_VAR
```

### AlarmyGlobal.typ - Global data types
```iecst
TYPE
	AlarmyVizu_typ : 	STRUCT
		PotvrdAlarmy : BOOL;
		ArchivaciaAlarmov : BOOL;
		ZobrazSymbolAlarmu : USINT;
		FarbaTlacitka_Alarmy : WSTRING[80];
	END_STRUCT;
END_TYPE
```

### AlarmyGlobal.var - Global variables
```iecst
VAR
	NastalaPorucha : BOOL;
	P1_AlarmyVizu : AlarmyVizu_typ;
	P2_AlarmyVizu : AlarmyVizu_typ;
	P34_AlarmyVizu : AlarmyVizu_typ;
	P1_PoruchaST1 : BOOL; (*Výtah*)
	P1_PoruchaST2 : BOOL; (*Šrobovanie*)
	P2_PoruchaST1 : BOOL; (*Zakladanie tesnenia*)
	P2_PoruchaST2 : BOOL; (*Skrutkovanie matic*)
	P2_PoruchaST3 : BOOL; (*Šrobovanie*)
	P2_PoruchaST4 : BOOL; (*Zvaranie*)
	P3_PoruchaST1 : BOOL;
	P3_PoruchaST2 : BOOL;
	P3_PoruchaST3 : BOOL;
	P4_PoruchaST1 : BOOL;
	P4_PoruchaST2 : BOOL;
	P4_PoruchaST3 : BOOL;
	P4_PoruchaST4 : BOOL;
	P1_Alarmy : ARRAY[100..199] OF BOOL;
	P2_Alarmy : ARRAY[200..299] OF BOOL;
	P34_Alarmy : ARRAY[300..499] OF BOOL;
	MpAlarmXCore_1 : MpAlarmXCore;
	MpAlarmXHistory_1 : MpAlarmXHistory;
END_VAR
```

### Program Logical/Alarmy/P1_Alarmy (IEC)
